// Mitsubishi GX Works2 project: LG Assembly 21-08-2019_F2   PLC: Q03UDV

PROGRAM MAIN
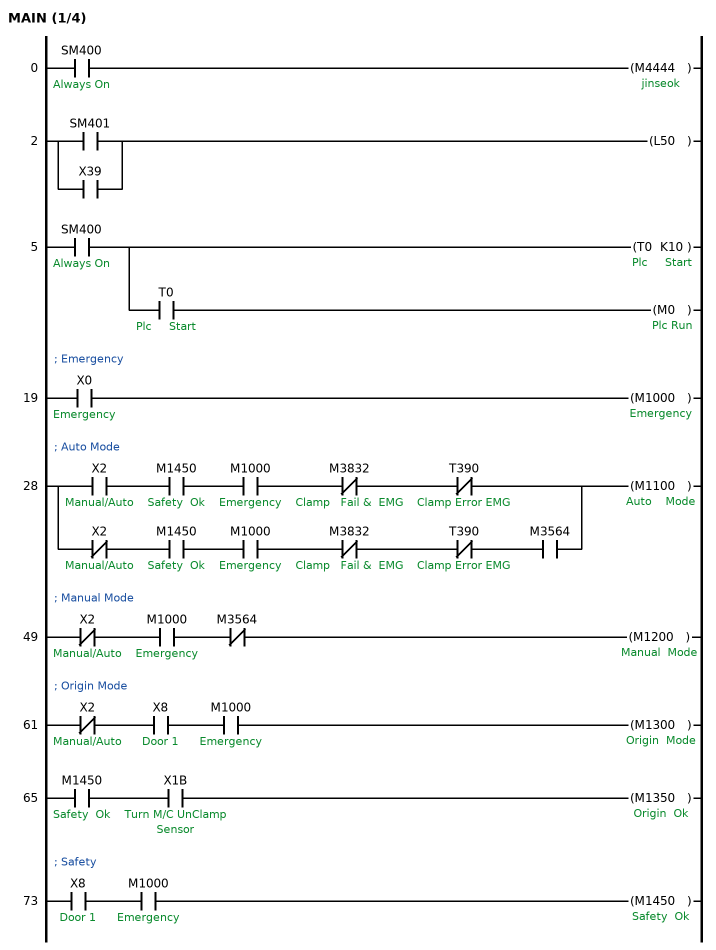
0     LD      SM400  ; Always On
      OUT     M4444  ; jinseok
2     LD      SM401
      OR      X39
      OUT     L50
5     LD      SM400  ; Always On
      OUT     T0 K10  ; Plc     Start
      AND     T0  ; Plc     Start
      OUT     M0  ; Plc Run
; Emergency
19    LD      X0  ; Emergency
      OUT     M1000  ; Emergency
; Auto Mode
28    LD      X2  ; Manual/Auto
      AND     M1450  ; Safety  Ok
      AND     M1000  ; Emergency
      ANI     M3832  ; Clamp   Fail &  EMG
      ANI     T390  ; Clamp Error EMG
      LDI     X2  ; Manual/Auto
      AND     M1450  ; Safety  Ok
      AND     M1000  ; Emergency
      ANI     M3832  ; Clamp   Fail &  EMG
      ANI     T390  ; Clamp Error EMG
      AND     M3564
      ORB
      OUT     M1100  ; Auto    Mode
; Manual Mode
49    LDI     X2  ; Manual/Auto
      AND     M1000  ; Emergency
      ANI     M3564
      OUT     M1200  ; Manual  Mode
; Origin Mode
61    LDI     X2  ; Manual/Auto
      AND     X8  ; Door 1
      AND     M1000  ; Emergency
      OUT     M1300  ; Origin  Mode
65    LD      M1450  ; Safety  Ok
      AND     X1B  ; Turn M/C UnClamp Sensor
      OUT     M1350  ; Origin  Ok
; Safety
73    LD      X8  ; Door 1
      AND     M1000  ; Emergency
      OUT     M1450  ; Safety  Ok
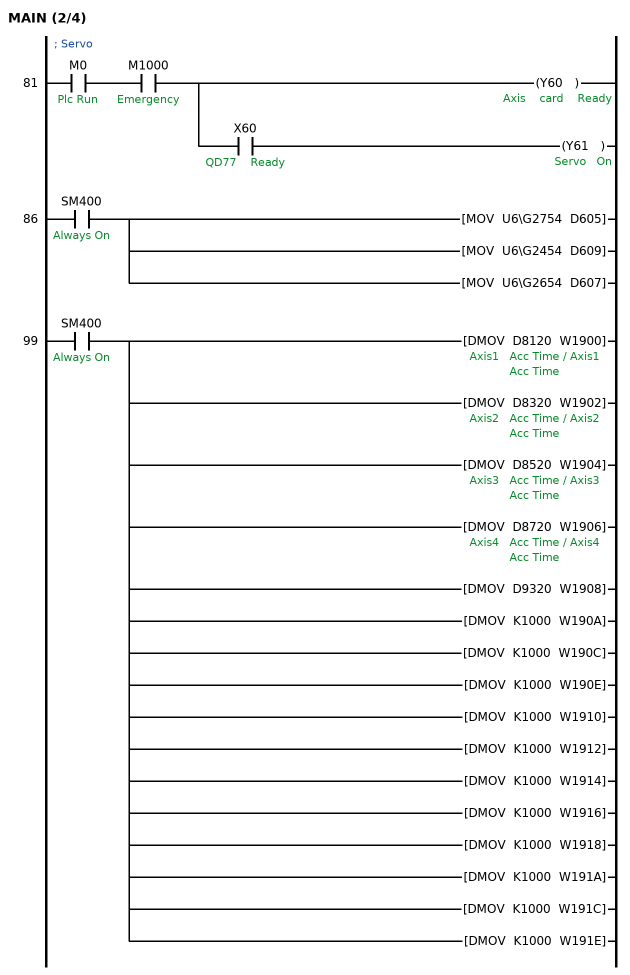
; Servo
81    LD      M0  ; Plc Run
      AND     M1000  ; Emergency
      OUT     Y60  ; Axis    card    Ready
      AND     X60  ; QD77    Ready
      OUT     Y61  ; Servo   On
86    LD      SM400  ; Always On
      MOV     U6\G2754 D605
      MOV     U6\G2454 D609
      MOV     U6\G2654 D607
99    LD      SM400  ; Always On
      DMOV    D8120 W1900  ; Axis1   Acc Time / Axis1   Acc Time
      DMOV    D8320 W1902  ; Axis2   Acc Time / Axis2   Acc Time
      DMOV    D8520 W1904  ; Axis3   Acc Time / Axis3   Acc Time
      DMOV    D8720 W1906  ; Axis4   Acc Time / Axis4   Acc Time
      DMOV    D9320 W1908
      DMOV    K1000 W190A
      DMOV    K1000 W190C
      DMOV    K1000 W190E
      DMOV    K1000 W1910
      DMOV    K1000 W1912
      DMOV    K1000 W1914
      DMOV    K1000 W1916
      DMOV    K1000 W1918
      DMOV    K1000 W191A
      DMOV    K1000 W191C
      DMOV    K1000 W191E
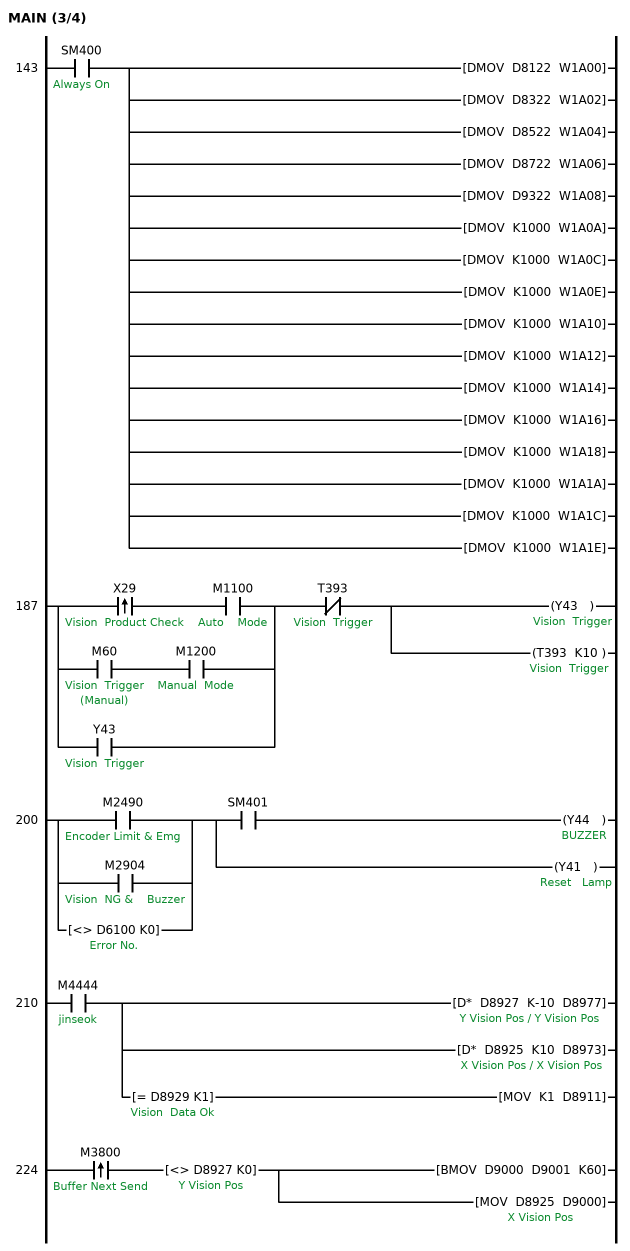
143   LD      SM400  ; Always On
      DMOV    D8122 W1A00
      DMOV    D8322 W1A02
      DMOV    D8522 W1A04
      DMOV    D8722 W1A06
      DMOV    D9322 W1A08
      DMOV    K1000 W1A0A
      DMOV    K1000 W1A0C
      DMOV    K1000 W1A0E
      DMOV    K1000 W1A10
      DMOV    K1000 W1A12
      DMOV    K1000 W1A14
      DMOV    K1000 W1A16
      DMOV    K1000 W1A18
      DMOV    K1000 W1A1A
      DMOV    K1000 W1A1C
      DMOV    K1000 W1A1E
187   LDP     X29  ; Vision  Product Check
      AND     M1100  ; Auto    Mode
      LD      M60  ; Vision  Trigger (Manual)
      AND     M1200  ; Manual  Mode
      ORB
      OR      Y43  ; Vision  Trigger
      ANI     T393  ; Vision  Trigger
      OUT     Y43  ; Vision  Trigger
      OUT     T393 K10  ; Vision  Trigger
200   LD      M2490  ; Encoder Limit & Emg
      OR      M2904  ; Vision  NG &    Buzzer
      OR<>    D6100 K0  ; Error No.
      MPS
      AND     SM401
      OUT     Y44  ; BUZZER
      MPP
      OUT     Y41  ; Reset   Lamp
210   LD      M4444  ; jinseok
      D*      D8927 K-10 D8977  ; Y Vision Pos / Y Vision Pos
      D*      D8925 K10 D8973  ; X Vision Pos / X Vision Pos
      AND=    D8929 K1  ; Vision  Data Ok
      MOV     K1 D8911
224   LDP     M3800  ; Buffer Next Send
      AND<>   D8927 K0  ; Y Vision Pos
      BMOV    D9000 D9001 K60
      MOV     D8925 D9000
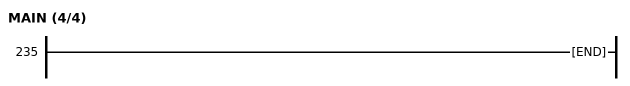
235   END
END_PROGRAM

PROGRAM ALARM
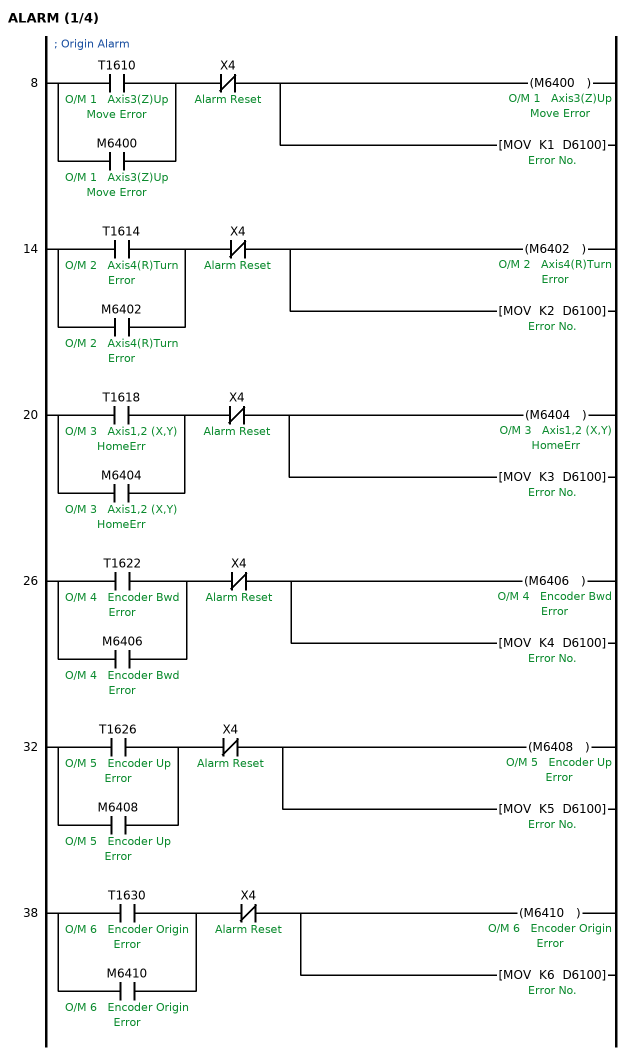
; Origin Alarm
8     LD      T1610  ; O/M 1   Axis3(Z)Up Move Error
      OR      M6400  ; O/M 1   Axis3(Z)Up Move Error
      ANI     X4  ; Alarm Reset
      OUT     M6400  ; O/M 1   Axis3(Z)Up Move Error
      MOV     K1 D6100  ; Error No.
14    LD      T1614  ; O/M 2   Axis4(R)Turn    Error
      OR      M6402  ; O/M 2   Axis4(R)Turn    Error
      ANI     X4  ; Alarm Reset
      OUT     M6402  ; O/M 2   Axis4(R)Turn    Error
      MOV     K2 D6100
20    LD      T1618  ; O/M 3   Axis1,2 (X,Y)   HomeErr
      OR      M6404  ; O/M 3   Axis1,2 (X,Y)   HomeErr
      ANI     X4  ; Alarm Reset
      OUT     M6404  ; O/M 3   Axis1,2 (X,Y)   HomeErr
      MOV     K3 D6100
26    LD      T1622  ; O/M 4   Encoder Bwd     Error
      OR      M6406  ; O/M 4   Encoder Bwd     Error
      ANI     X4  ; Alarm Reset
      OUT     M6406  ; O/M 4   Encoder Bwd     Error
      MOV     K4 D6100
32    LD      T1626  ; O/M 5   Encoder Up      Error
      OR      M6408  ; O/M 5   Encoder Up      Error
      ANI     X4  ; Alarm Reset
      OUT     M6408  ; O/M 5   Encoder Up      Error
      MOV     K5 D6100
38    LD      T1630  ; O/M 6   Encoder Origin  Error
      OR      M6410  ; O/M 6   Encoder Origin  Error
      ANI     X4  ; Alarm Reset
      OUT     M6410  ; O/M 6   Encoder Origin  Error
      MOV     K6 D6100
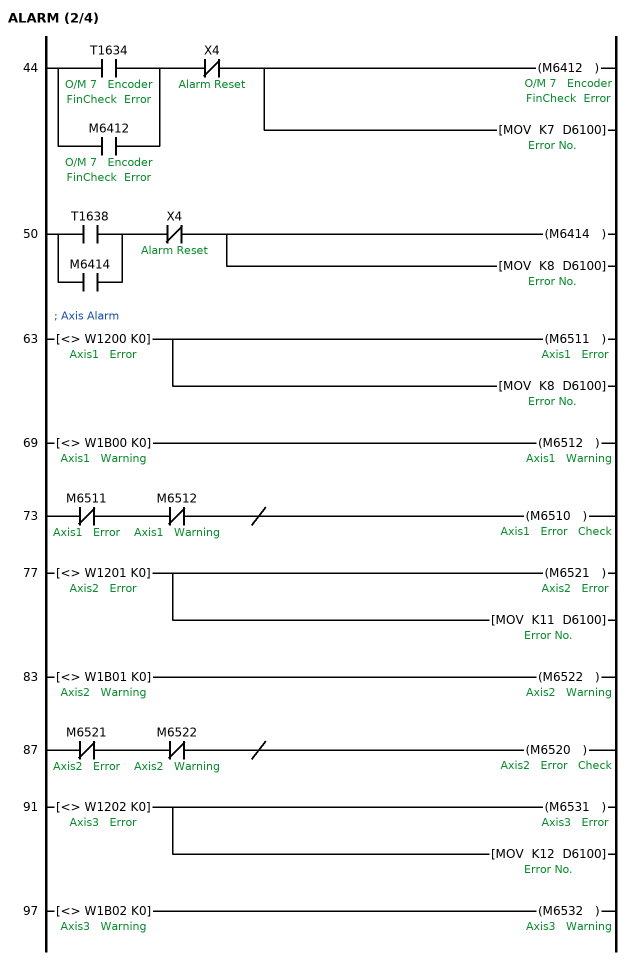
44    LD      T1634  ; O/M 7   Encoder FinCheck  Error
      OR      M6412  ; O/M 7   Encoder FinCheck  Error
      ANI     X4  ; Alarm Reset
      OUT     M6412  ; O/M 7   Encoder FinCheck  Error
      MOV     K7 D6100
50    LD      T1638
      OR      M6414
      ANI     X4  ; Alarm Reset
      OUT     M6414
      MOV     K8 D6100
; Axis Alarm
63    LD<>    W1200 K0  ; Axis1   Error
      OUT     M6511  ; Axis1   Error
      MOV     K8 D6100
69    LD<>    W1B00 K0  ; Axis1   Warning
      OUT     M6512  ; Axis1   Warning
73    LDI     M6511  ; Axis1   Error
      ANI     M6512  ; Axis1   Warning
      INV
      OUT     M6510  ; Axis1   Error   Check
77    LD<>    W1201 K0  ; Axis2   Error
      OUT     M6521  ; Axis2   Error
      MOV     K11 D6100
83    LD<>    W1B01 K0  ; Axis2   Warning
      OUT     M6522  ; Axis2   Warning
87    LDI     M6521  ; Axis2   Error
      ANI     M6522  ; Axis2   Warning
      INV
      OUT     M6520  ; Axis2   Error   Check
91    LD<>    W1202 K0  ; Axis3   Error
      OUT     M6531  ; Axis3   Error
      MOV     K12 D6100
97    LD<>    W1B02 K0  ; Axis3   Warning
      OUT     M6532  ; Axis3   Warning
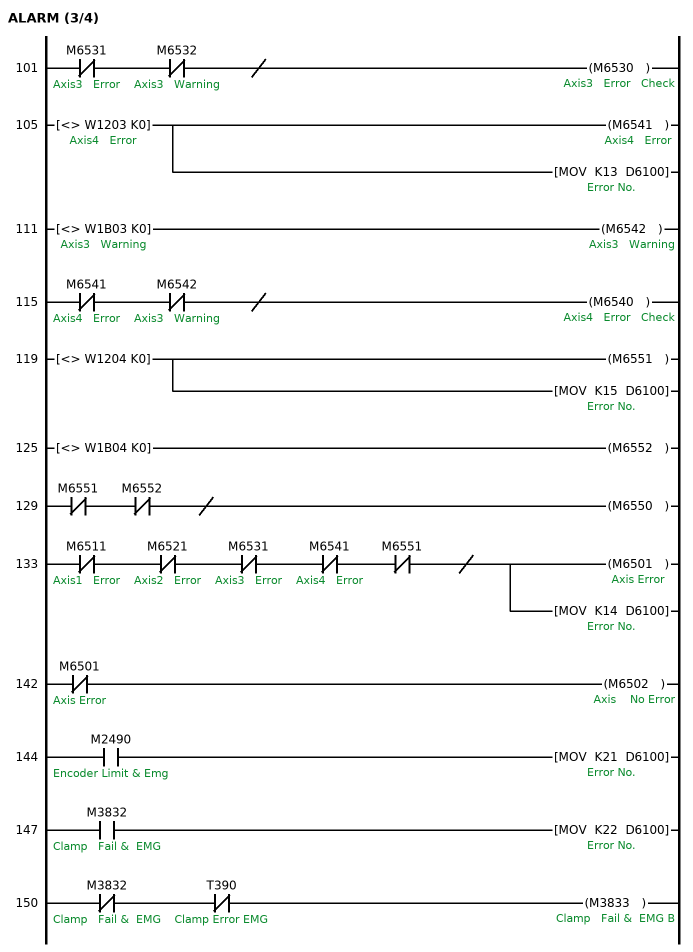
101   LDI     M6531  ; Axis3   Error
      ANI     M6532  ; Axis3   Warning
      INV
      OUT     M6530  ; Axis3   Error   Check
105   LD<>    W1203 K0  ; Axis4   Error
      OUT     M6541  ; Axis4   Error
      MOV     K13 D6100
111   LD<>    W1B03 K0  ; Axis3   Warning
      OUT     M6542  ; Axis3   Warning
115   LDI     M6541  ; Axis4   Error
      ANI     M6542  ; Axis3   Warning
      INV
      OUT     M6540  ; Axis4   Error   Check
119   LD<>    W1204 K0
      OUT     M6551
      MOV     K15 D6100
125   LD<>    W1B04 K0
      OUT     M6552
129   LDI     M6551
      ANI     M6552
      INV
      OUT     M6550
133   LDI     M6511  ; Axis1   Error
      ANI     M6521  ; Axis2   Error
      ANI     M6531  ; Axis3   Error
      ANI     M6541  ; Axis4   Error
      ANI     M6551
      INV
      OUT     M6501  ; Axis Error
      MOV     K14 D6100
142   LDI     M6501  ; Axis Error
      OUT     M6502  ; Axis    No Error
144   LD      M2490  ; Encoder Limit & Emg
      MOV     K21 D6100
147   LD      M3832  ; Clamp   Fail &  EMG
      MOV     K22 D6100
150   LDI     M3832  ; Clamp   Fail &  EMG
      ANI     T390  ; Clamp Error EMG
      OUT     M3833  ; Clamp   Fail &  EMG B
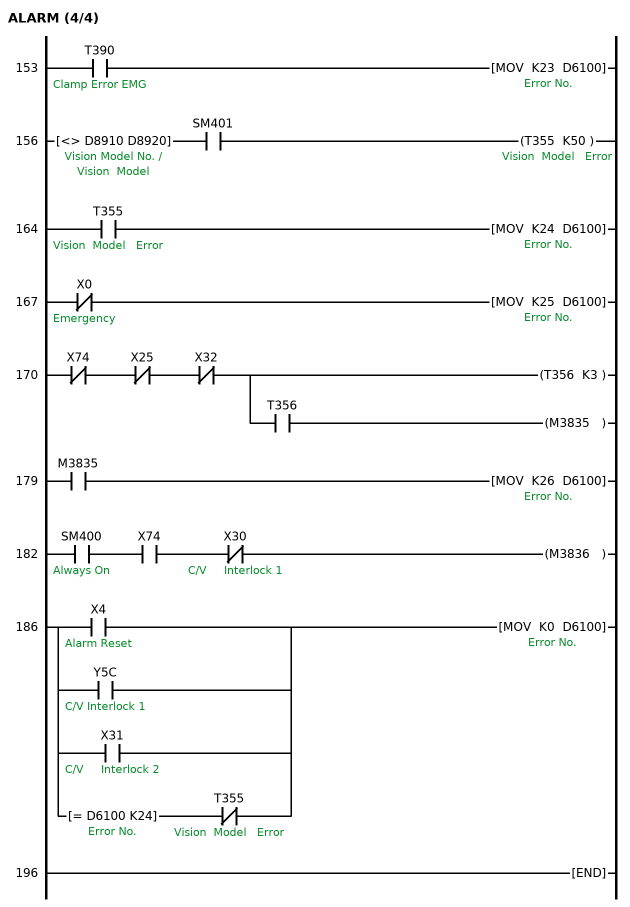
153   LD      T390  ; Clamp Error EMG
      MOV     K23 D6100
156   LD<>    D8910 D8920  ; Vision Model No. / Vision  Model
      AND     SM401
      OUT     T355 K50  ; Vision  Model   Error
164   LD      T355  ; Vision  Model   Error
      MOV     K24 D6100
167   LDI     X0  ; Emergency
      MOV     K25 D6100
170   LDI     X74
      ANI     X25
      ANI     X32
      OUT     T356 K3
      AND     T356
      OUT     M3835
179   LD      M3835
      MOV     K26 D6100
182   LD      SM400  ; Always On
      AND     X74
      ANI     X30  ; C/V     Interlock 1
      OUT     M3836
186   LD      X4  ; Alarm Reset
      OR      Y5C  ; C/V Interlock 1
      OR      X31  ; C/V     Interlock 2
      LD=     D6100 K24  ; Error No.
      ANI     T355  ; Vision  Model   Error
      ORB
      MOV     K0 D6100
196   END
END_PROGRAM

PROGRAM AUTO
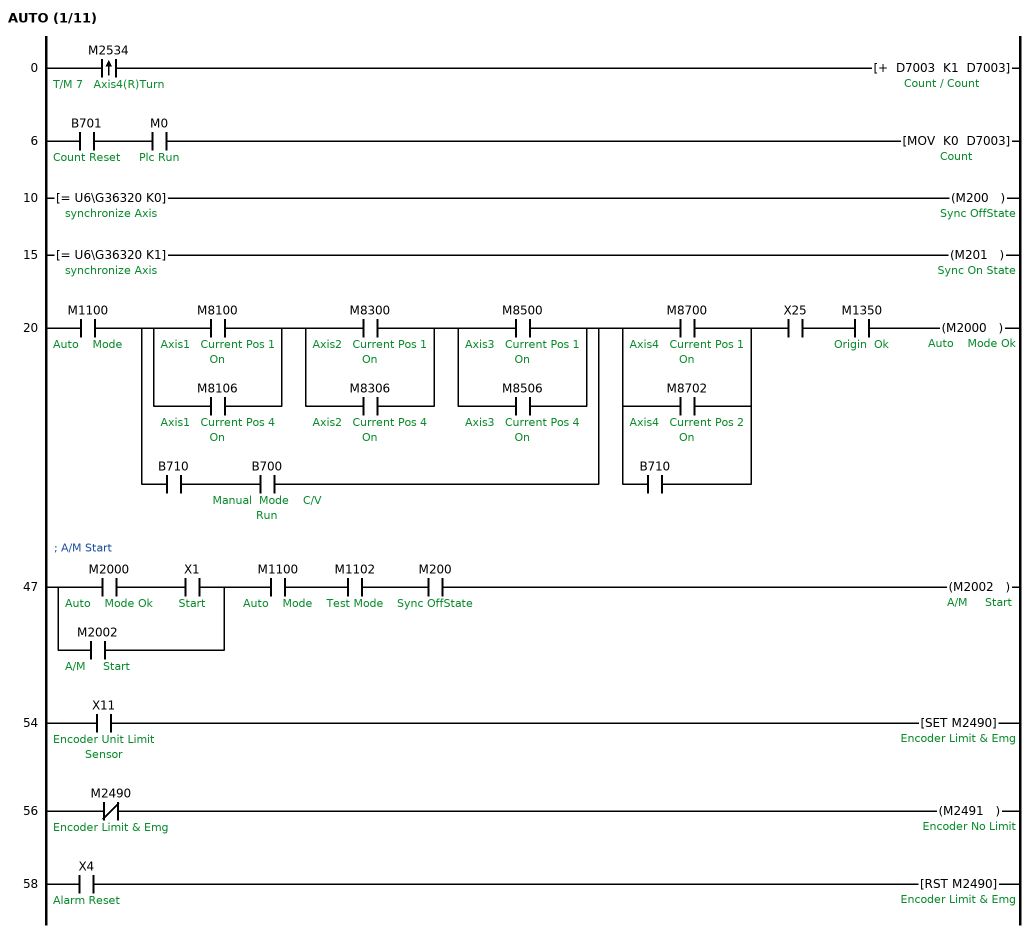
0     LDP     M2534  ; T/M 7   Axis4(R)Turn
      +       D7003 K1 D7003  ; Count
6     LD      B701  ; Count Reset
      AND     M0  ; Plc Run
      MOV     K0 D7003
10    LD=     U6\G36320 K0  ; synchronize Axis
      OUT     M200  ; Sync OffState
15    LD=     U6\G36320 K1  ; synchronize Axis
      OUT     M201  ; Sync On State
20    LD      M1100  ; Auto    Mode
      LD      M8100  ; Axis1   Current Pos 1 On
      OR      M8106  ; Axis1   Current Pos 4 On
      LD      M8300  ; Axis2   Current Pos 1 On
      OR      M8306  ; Axis2   Current Pos 4 On
      ANB
      LD      M8500  ; Axis3   Current Pos 1 On
      OR      M8506  ; Axis3   Current Pos 4 On
      ANB
      LD      B710
      AND     B700  ; Manual  Mode    C/V Run
      ORB
      ANB
      LD      M8700  ; Axis4   Current Pos 1 On
      OR      M8702  ; Axis4   Current Pos 2 On
      OR      B710
      ANB
      AND     X25
      AND     M1350  ; Origin  Ok
      OUT     M2000  ; Auto    Mode Ok
; A/M Start
47    LD      M2000  ; Auto    Mode Ok
      AND     X1  ; Start
      OR      M2002  ; A/M     Start
      AND     M1100  ; Auto    Mode
      AND     M1102  ; Test Mode
      AND     M200  ; Sync OffState
      OUT     M2002  ; A/M     Start
54    LD      X11  ; Encoder Unit Limit Sensor
      SET     M2490  ; Encoder Limit & Emg
56    LDI     M2490  ; Encoder Limit & Emg
      OUT     M2491  ; Encoder No Limit
58    LD      X4  ; Alarm Reset
      RST     M2490  ; Encoder Limit & Emg
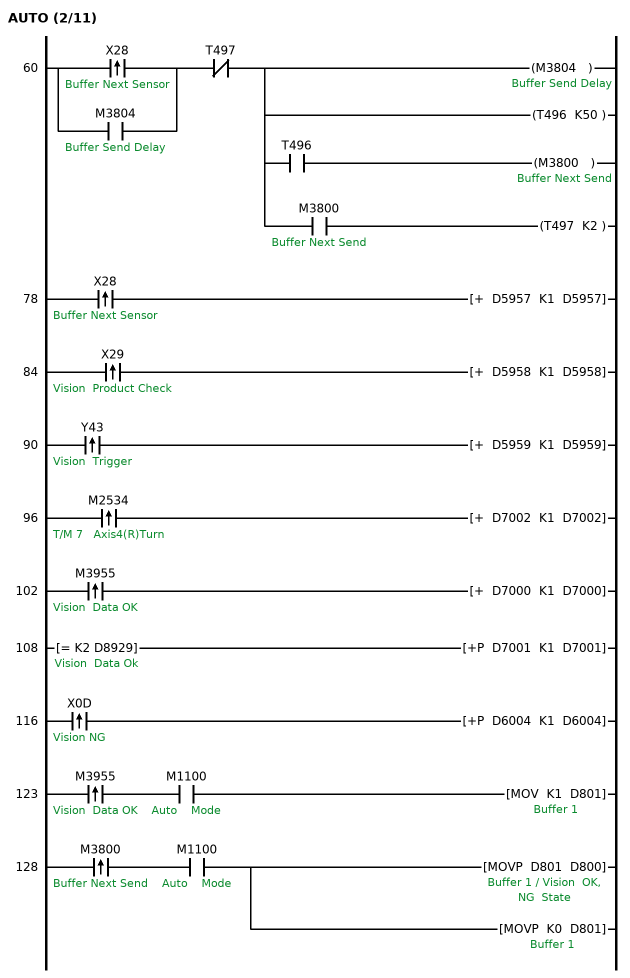
60    LDP     X28  ; Buffer Next Sensor
      OR      M3804  ; Buffer Send Delay
      ANI     T497
      OUT     M3804  ; Buffer Send Delay
      OUT     T496 K50
      MPS
      AND     T496
      OUT     M3800  ; Buffer Next Send
      MPP
      AND     M3800  ; Buffer Next Send
      OUT     T497 K2
78    LDP     X28  ; Buffer Next Sensor
      +       D5957 K1 D5957
84    LDP     X29  ; Vision  Product Check
      +       D5958 K1 D5958
90    LDP     Y43  ; Vision  Trigger
      +       D5959 K1 D5959
96    LDP     M2534  ; T/M 7   Axis4(R)Turn
      +       D7002 K1 D7002
102   LDP     M3955  ; Vision  Data OK
      +       D7000 K1 D7000
108   LD=     K2 D8929  ; Vision  Data Ok
      +P      D7001 K1 D7001
116   LDP     X0D  ; Vision NG
      +P      D6004 K1 D6004
123   LDP     M3955  ; Vision  Data OK
      AND     M1100  ; Auto    Mode
      MOV     K1 D801  ; Buffer 1
128   LDP     M3800  ; Buffer Next Send
      AND     M1100  ; Auto    Mode
      MOVP    D801 D800  ; Vision  OK, NG  State
      MOVP    K0 D801
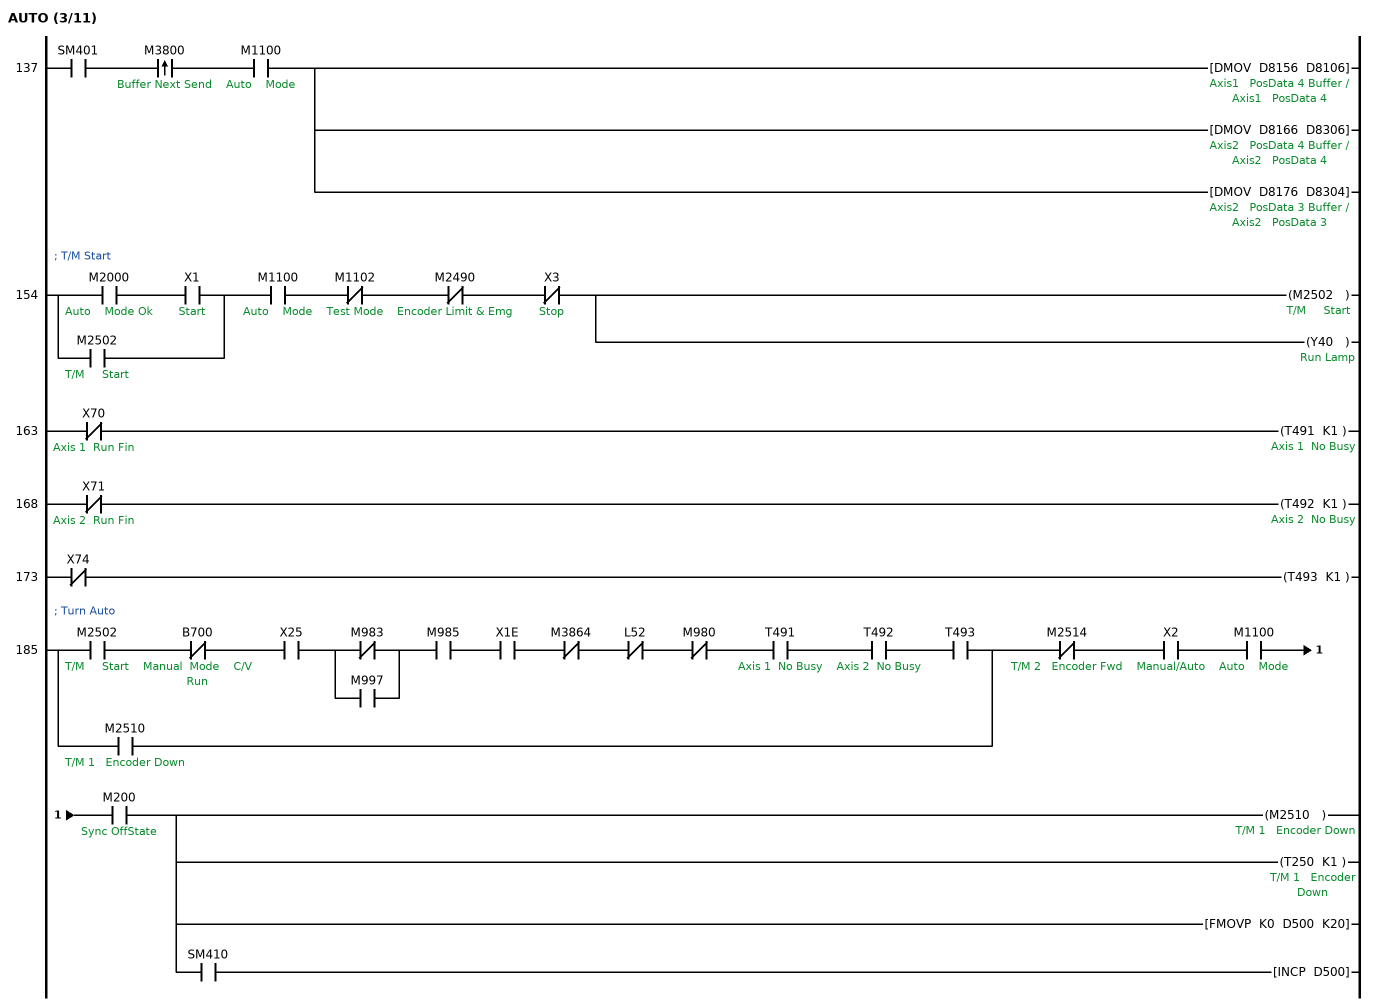
137   LD      SM401
      ANDP    M3800  ; Buffer Next Send
      AND     M1100  ; Auto    Mode
      DMOV    D8156 D8106  ; Axis1   PosData 4 Buffer / Axis1   PosData 4
      DMOV    D8166 D8306  ; Axis2   PosData 4 Buffer / Axis2   PosData 4
      DMOV    D8176 D8304  ; Axis2   PosData 3 Buffer / Axis2   PosData 3
; T/M Start
154   LD      M2000  ; Auto    Mode Ok
      AND     X1  ; Start
      OR      M2502  ; T/M     Start
      AND     M1100  ; Auto    Mode
      ANI     M1102  ; Test Mode
      ANI     M2490  ; Encoder Limit & Emg
      ANI     X3  ; Stop
      OUT     M2502  ; T/M     Start
      OUT     Y40  ; Run Lamp
163   LDI     X70  ; Axis 1  Run Fin
      OUT     T491 K1  ; Axis 1  No Busy
168   LDI     X71  ; Axis 2  Run Fin
      OUT     T492 K1  ; Axis 2  No Busy
173   LDI     X74
      OUT     T493 K1
; Turn Auto
185   LD      M2502  ; T/M     Start
      ANI     B700  ; Manual  Mode    C/V Run
      AND     X25
      LDI     M983
      OR      M997
      ANB
      AND     M985
      AND     X1E
      ANI     M3864
      ANI     L52
      ANI     M980
      AND     T491  ; Axis 1  No Busy
      AND     T492  ; Axis 2  No Busy
      AND     T493
      OR      M2510  ; T/M 1   Encoder Down
      ANI     M2514  ; T/M 2   Encoder Fwd
      AND     X2  ; Manual/Auto
      AND     M1100  ; Auto    Mode
      AND     M200  ; Sync OffState
      OUT     M2510  ; T/M 1   Encoder Down
      OUT     T250 K1  ; T/M 1   Encoder Down
      FMOVP   K0 D500 K20
      AND     SM410
      INCP    D500
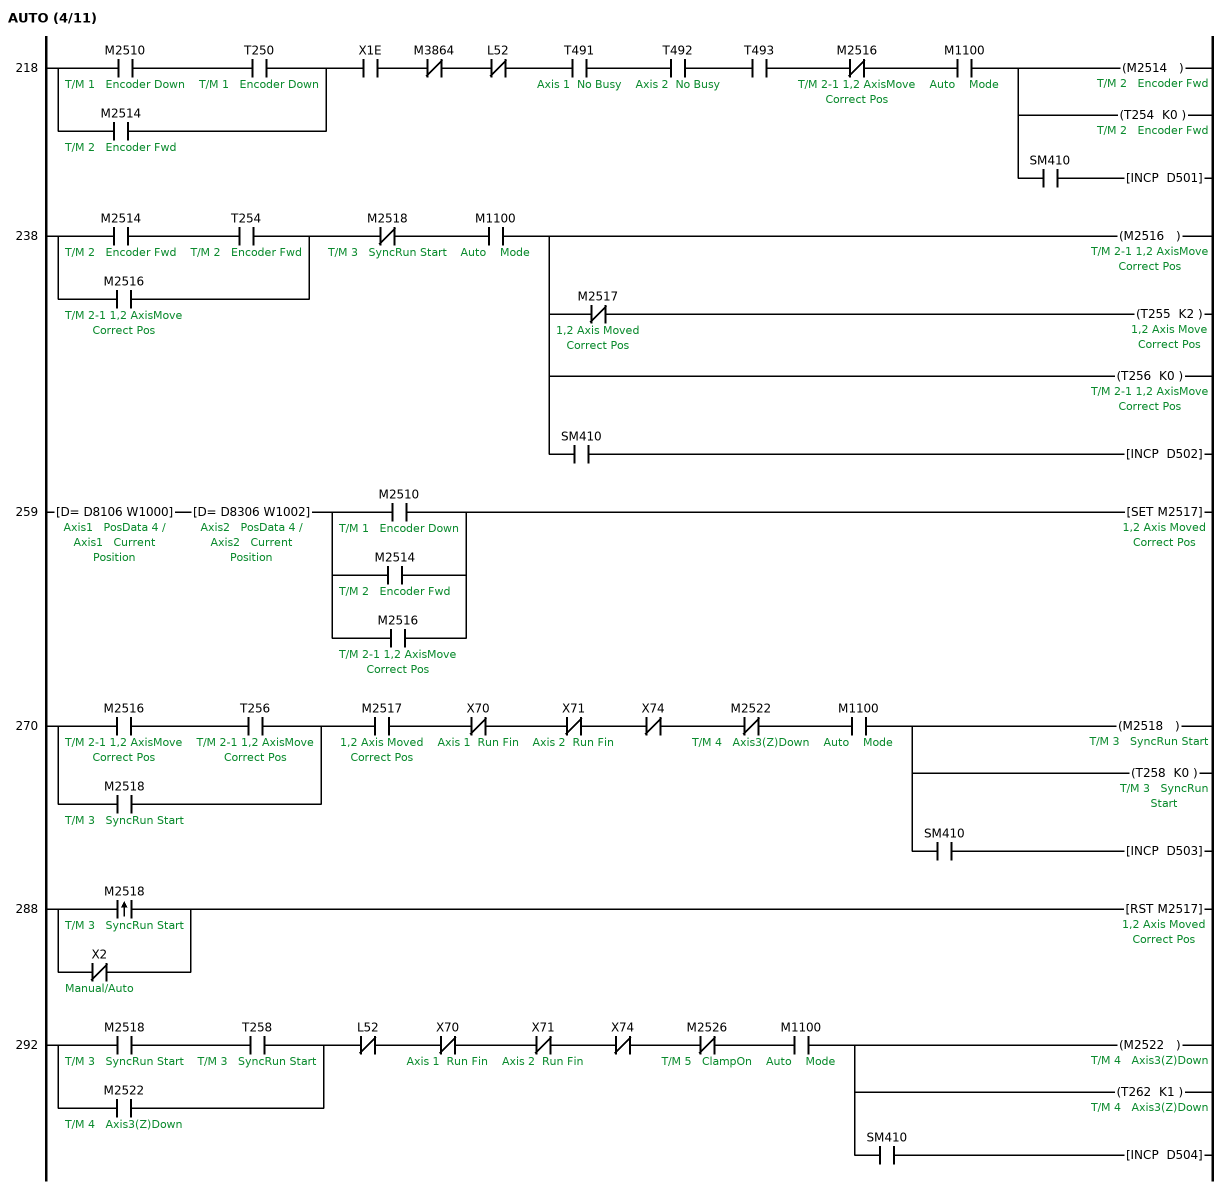
218   LD      M2510  ; T/M 1   Encoder Down
      AND     T250  ; T/M 1   Encoder Down
      OR      M2514  ; T/M 2   Encoder Fwd
      AND     X1E
      ANI     M3864
      ANI     L52
      AND     T491  ; Axis 1  No Busy
      AND     T492  ; Axis 2  No Busy
      AND     T493
      ANI     M2516  ; T/M 2-1 1,2 AxisMove Correct Pos
      AND     M1100  ; Auto    Mode
      OUT     M2514  ; T/M 2   Encoder Fwd
      OUT     T254 K0  ; T/M 2   Encoder Fwd
      AND     SM410
      INCP    D501
238   LD      M2514  ; T/M 2   Encoder Fwd
      AND     T254  ; T/M 2   Encoder Fwd
      OR      M2516  ; T/M 2-1 1,2 AxisMove Correct Pos
      ANI     M2518  ; T/M 3   SyncRun Start
      AND     M1100  ; Auto    Mode
      OUT     M2516  ; T/M 2-1 1,2 AxisMove Correct Pos
      MPS
      ANI     M2517  ; 1,2 Axis Moved Correct Pos
      OUT     T255 K2  ; 1,2 Axis Move Correct Pos
      MPP
      OUT     T256 K0  ; T/M 2-1 1,2 AxisMove Correct Pos
      AND     SM410
      INCP    D502
259   LDD=    D8106 W1000  ; Axis1   PosData 4 / Axis1   Current Position
      ANDD=   D8306 W1002  ; Axis2   PosData 4 / Axis2   Current Position
      LD      M2510  ; T/M 1   Encoder Down
      OR      M2514  ; T/M 2   Encoder Fwd
      OR      M2516  ; T/M 2-1 1,2 AxisMove Correct Pos
      ANB
      SET     M2517  ; 1,2 Axis Moved Correct Pos
270   LD      M2516  ; T/M 2-1 1,2 AxisMove Correct Pos
      AND     T256  ; T/M 2-1 1,2 AxisMove Correct Pos
      OR      M2518  ; T/M 3   SyncRun Start
      AND     M2517  ; 1,2 Axis Moved Correct Pos
      ANI     X70  ; Axis 1  Run Fin
      ANI     X71  ; Axis 2  Run Fin
      ANI     X74
      ANI     M2522  ; T/M 4   Axis3(Z)Down
      AND     M1100  ; Auto    Mode
      OUT     M2518  ; T/M 3   SyncRun Start
      OUT     T258 K0  ; T/M 3   SyncRun Start
      AND     SM410
      INCP    D503
288   LDP     M2518  ; T/M 3   SyncRun Start
      ORI     X2  ; Manual/Auto
      RST     M2517  ; 1,2 Axis Moved Correct Pos
292   LD      M2518  ; T/M 3   SyncRun Start
      AND     T258  ; T/M 3   SyncRun Start
      OR      M2522  ; T/M 4   Axis3(Z)Down
      ANI     L52
      ANI     X70  ; Axis 1  Run Fin
      ANI     X71  ; Axis 2  Run Fin
      ANI     X74
      ANI     M2526  ; T/M 5   ClampOn
      AND     M1100  ; Auto    Mode
      OUT     M2522  ; T/M 4   Axis3(Z)Down
      OUT     T262 K1  ; T/M 4   Axis3(Z)Down
      AND     SM410
      INCP    D504
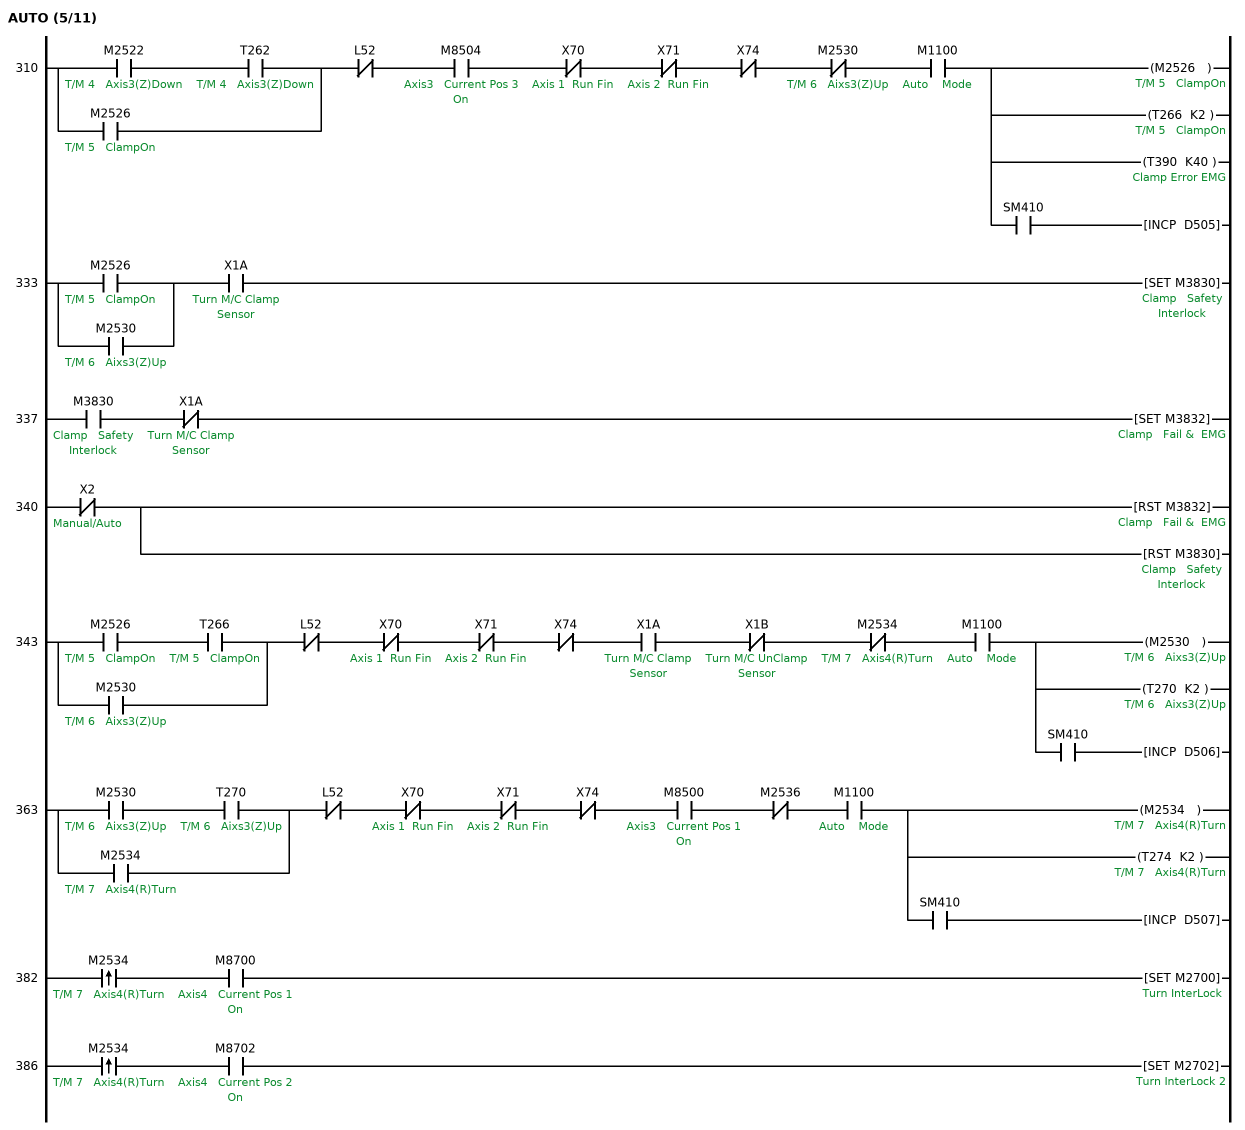
310   LD      M2522  ; T/M 4   Axis3(Z)Down
      AND     T262  ; T/M 4   Axis3(Z)Down
      OR      M2526  ; T/M 5   ClampOn
      ANI     L52
      AND     M8504  ; Axis3   Current Pos 3 On
      ANI     X70  ; Axis 1  Run Fin
      ANI     X71  ; Axis 2  Run Fin
      ANI     X74
      ANI     M2530  ; T/M 6   Aixs3(Z)Up
      AND     M1100  ; Auto    Mode
      OUT     M2526  ; T/M 5   ClampOn
      OUT     T266 K2  ; T/M 5   ClampOn
      OUT     T390 K40  ; Clamp Error EMG
      AND     SM410
      INCP    D505
333   LD      M2526  ; T/M 5   ClampOn
      OR      M2530  ; T/M 6   Aixs3(Z)Up
      AND     X1A  ; Turn M/C Clamp Sensor
      SET     M3830  ; Clamp   Safety  Interlock
337   LD      M3830  ; Clamp   Safety  Interlock
      ANI     X1A  ; Turn M/C Clamp Sensor
      SET     M3832  ; Clamp   Fail &  EMG
340   LDI     X2  ; Manual/Auto
      RST     M3832  ; Clamp   Fail &  EMG
      RST     M3830  ; Clamp   Safety  Interlock
343   LD      M2526  ; T/M 5   ClampOn
      AND     T266  ; T/M 5   ClampOn
      OR      M2530  ; T/M 6   Aixs3(Z)Up
      ANI     L52
      ANI     X70  ; Axis 1  Run Fin
      ANI     X71  ; Axis 2  Run Fin
      ANI     X74
      AND     X1A  ; Turn M/C Clamp Sensor
      ANI     X1B  ; Turn M/C UnClamp Sensor
      ANI     M2534  ; T/M 7   Axis4(R)Turn
      AND     M1100  ; Auto    Mode
      OUT     M2530  ; T/M 6   Aixs3(Z)Up
      OUT     T270 K2  ; T/M 6   Aixs3(Z)Up
      AND     SM410
      INCP    D506
363   LD      M2530  ; T/M 6   Aixs3(Z)Up
      AND     T270  ; T/M 6   Aixs3(Z)Up
      OR      M2534  ; T/M 7   Axis4(R)Turn
      ANI     L52
      ANI     X70  ; Axis 1  Run Fin
      ANI     X71  ; Axis 2  Run Fin
      ANI     X74
      AND     M8500  ; Axis3   Current Pos 1 On
      ANI     M2536
      AND     M1100  ; Auto    Mode
      OUT     M2534  ; T/M 7   Axis4(R)Turn
      OUT     T274 K2  ; T/M 7   Axis4(R)Turn
      AND     SM410
      INCP    D507
382   LDP     M2534  ; T/M 7   Axis4(R)Turn
      AND     M8700  ; Axis4   Current Pos 1 On
      SET     M2700  ; Turn InterLock
386   LDP     M2534  ; T/M 7   Axis4(R)Turn
      AND     M8702  ; Axis4   Current Pos 2 On
      SET     M2702  ; Turn InterLock 2
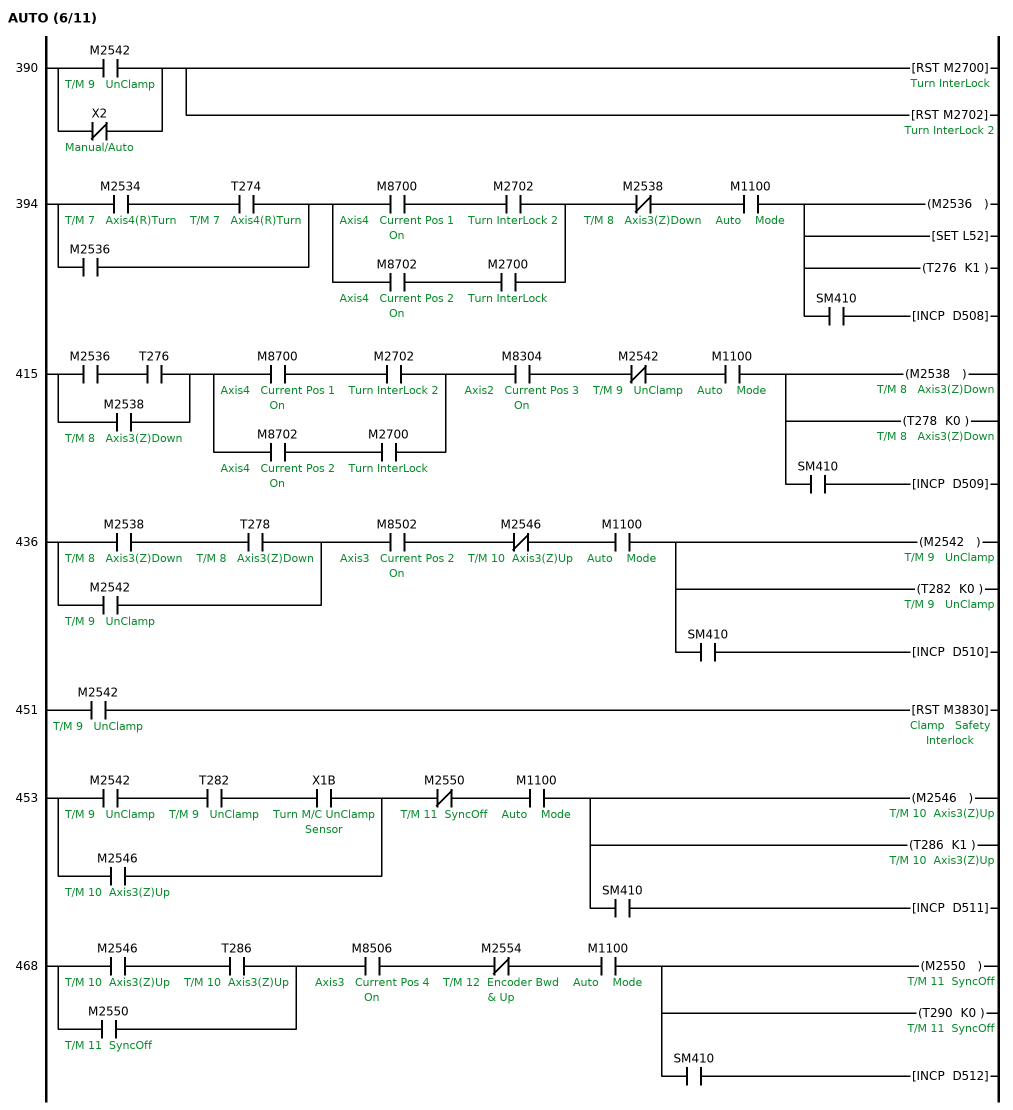
390   LD      M2542  ; T/M 9   UnClamp
      ORI     X2  ; Manual/Auto
      RST     M2700  ; Turn InterLock
      RST     M2702  ; Turn InterLock 2
394   LD      M2534  ; T/M 7   Axis4(R)Turn
      AND     T274  ; T/M 7   Axis4(R)Turn
      OR      M2536
      LD      M8700  ; Axis4   Current Pos 1 On
      AND     M2702  ; Turn InterLock 2
      LD      M8702  ; Axis4   Current Pos 2 On
      AND     M2700  ; Turn InterLock
      ORB
      ANB
      ANI     M2538  ; T/M 8   Axis3(Z)Down
      AND     M1100  ; Auto    Mode
      OUT     M2536
      SET     L52
      OUT     T276 K1
      AND     SM410
      INCP    D508
415   LD      M2536
      AND     T276
      OR      M2538  ; T/M 8   Axis3(Z)Down
      LD      M8700  ; Axis4   Current Pos 1 On
      AND     M2702  ; Turn InterLock 2
      LD      M8702  ; Axis4   Current Pos 2 On
      AND     M2700  ; Turn InterLock
      ORB
      ANB
      AND     M8304  ; Axis2   Current Pos 3 On
      ANI     M2542  ; T/M 9   UnClamp
      AND     M1100  ; Auto    Mode
      OUT     M2538  ; T/M 8   Axis3(Z)Down
      OUT     T278 K0  ; T/M 8   Axis3(Z)Down
      AND     SM410
      INCP    D509
436   LD      M2538  ; T/M 8   Axis3(Z)Down
      AND     T278  ; T/M 8   Axis3(Z)Down
      OR      M2542  ; T/M 9   UnClamp
      AND     M8502  ; Axis3   Current Pos 2 On
      ANI     M2546  ; T/M 10  Axis3(Z)Up
      AND     M1100  ; Auto    Mode
      OUT     M2542  ; T/M 9   UnClamp
      OUT     T282 K0  ; T/M 9   UnClamp
      AND     SM410
      INCP    D510
451   LD      M2542  ; T/M 9   UnClamp
      RST     M3830  ; Clamp   Safety  Interlock
453   LD      M2542  ; T/M 9   UnClamp
      AND     T282  ; T/M 9   UnClamp
      AND     X1B  ; Turn M/C UnClamp Sensor
      OR      M2546  ; T/M 10  Axis3(Z)Up
      ANI     M2550  ; T/M 11  SyncOff
      AND     M1100  ; Auto    Mode
      OUT     M2546  ; T/M 10  Axis3(Z)Up
      OUT     T286 K1  ; T/M 10  Axis3(Z)Up
      AND     SM410
      INCP    D511
468   LD      M2546  ; T/M 10  Axis3(Z)Up
      AND     T286  ; T/M 10  Axis3(Z)Up
      OR      M2550  ; T/M 11  SyncOff
      AND     M8506  ; Axis3   Current Pos 4 On
      ANI     M2554  ; T/M 12  Encoder Bwd & Up
      AND     M1100  ; Auto    Mode
      OUT     M2550  ; T/M 11  SyncOff
      OUT     T290 K0  ; T/M 11  SyncOff
      AND     SM410
      INCP    D512
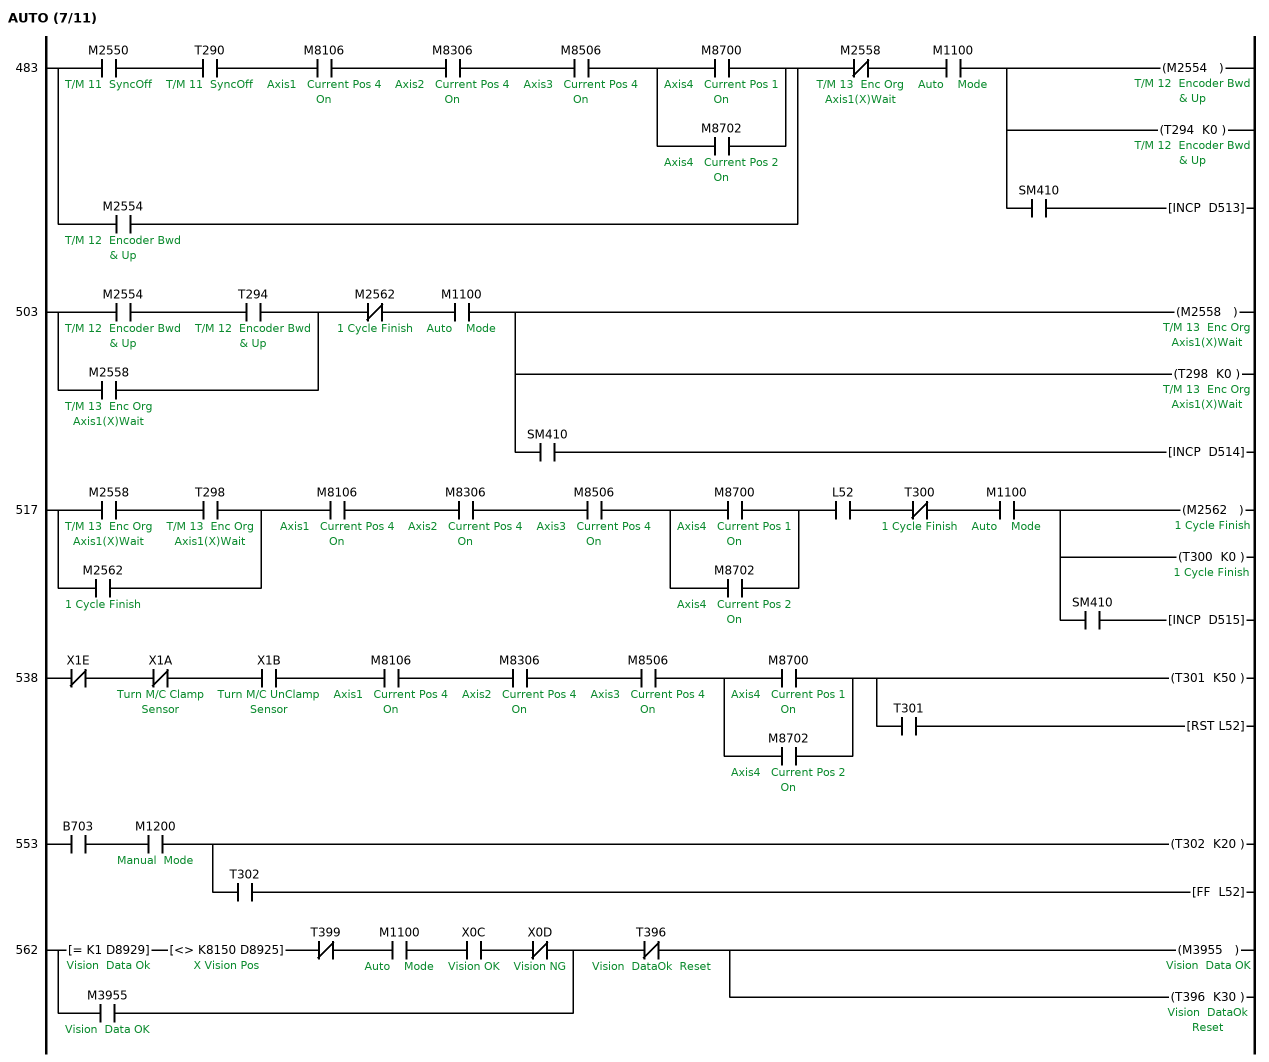
483   LD      M2550  ; T/M 11  SyncOff
      AND     T290  ; T/M 11  SyncOff
      AND     M8106  ; Axis1   Current Pos 4 On
      AND     M8306  ; Axis2   Current Pos 4 On
      AND     M8506  ; Axis3   Current Pos 4 On
      LD      M8700  ; Axis4   Current Pos 1 On
      OR      M8702  ; Axis4   Current Pos 2 On
      ANB
      OR      M2554  ; T/M 12  Encoder Bwd & Up
      ANI     M2558  ; T/M 13  Enc Org Axis1(X)Wait
      AND     M1100  ; Auto    Mode
      OUT     M2554  ; T/M 12  Encoder Bwd & Up
      OUT     T294 K0  ; T/M 12  Encoder Bwd & Up
      AND     SM410
      INCP    D513
503   LD      M2554  ; T/M 12  Encoder Bwd & Up
      AND     T294  ; T/M 12  Encoder Bwd & Up
      OR      M2558  ; T/M 13  Enc Org Axis1(X)Wait
      ANI     M2562  ; 1 Cycle Finish
      AND     M1100  ; Auto    Mode
      OUT     M2558  ; T/M 13  Enc Org Axis1(X)Wait
      OUT     T298 K0  ; T/M 13  Enc Org Axis1(X)Wait
      AND     SM410
      INCP    D514
517   LD      M2558  ; T/M 13  Enc Org Axis1(X)Wait
      AND     T298  ; T/M 13  Enc Org Axis1(X)Wait
      OR      M2562  ; 1 Cycle Finish
      AND     M8106  ; Axis1   Current Pos 4 On
      AND     M8306  ; Axis2   Current Pos 4 On
      AND     M8506  ; Axis3   Current Pos 4 On
      LD      M8700  ; Axis4   Current Pos 1 On
      OR      M8702  ; Axis4   Current Pos 2 On
      ANB
      AND     L52
      ANI     T300  ; 1 Cycle Finish
      AND     M1100  ; Auto    Mode
      OUT     M2562  ; 1 Cycle Finish
      OUT     T300 K0  ; 1 Cycle Finish
      AND     SM410
      INCP    D515
538   LDI     X1E
      ANI     X1A  ; Turn M/C Clamp Sensor
      AND     X1B  ; Turn M/C UnClamp Sensor
      AND     M8106  ; Axis1   Current Pos 4 On
      AND     M8306  ; Axis2   Current Pos 4 On
      AND     M8506  ; Axis3   Current Pos 4 On
      LD      M8700  ; Axis4   Current Pos 1 On
      OR      M8702  ; Axis4   Current Pos 2 On
      ANB
      OUT     T301 K50
      AND     T301
      RST     L52
553   LD      B703
      AND     M1200  ; Manual  Mode
      OUT     T302 K20
      AND     T302
      FF      L52
562   LD=     K1 D8929  ; Vision  Data Ok
      AND<>   K8150 D8925  ; X Vision Pos
      ANI     T399
      AND     M1100  ; Auto    Mode
      AND     X0C  ; Vision OK
      ANI     X0D  ; Vision NG
      OR      M3955  ; Vision  Data OK
      ANI     T396  ; Vision  DataOk  Reset
      OUT     M3955  ; Vision  Data OK
      OUT     T396 K30  ; Vision  DataOk  Reset
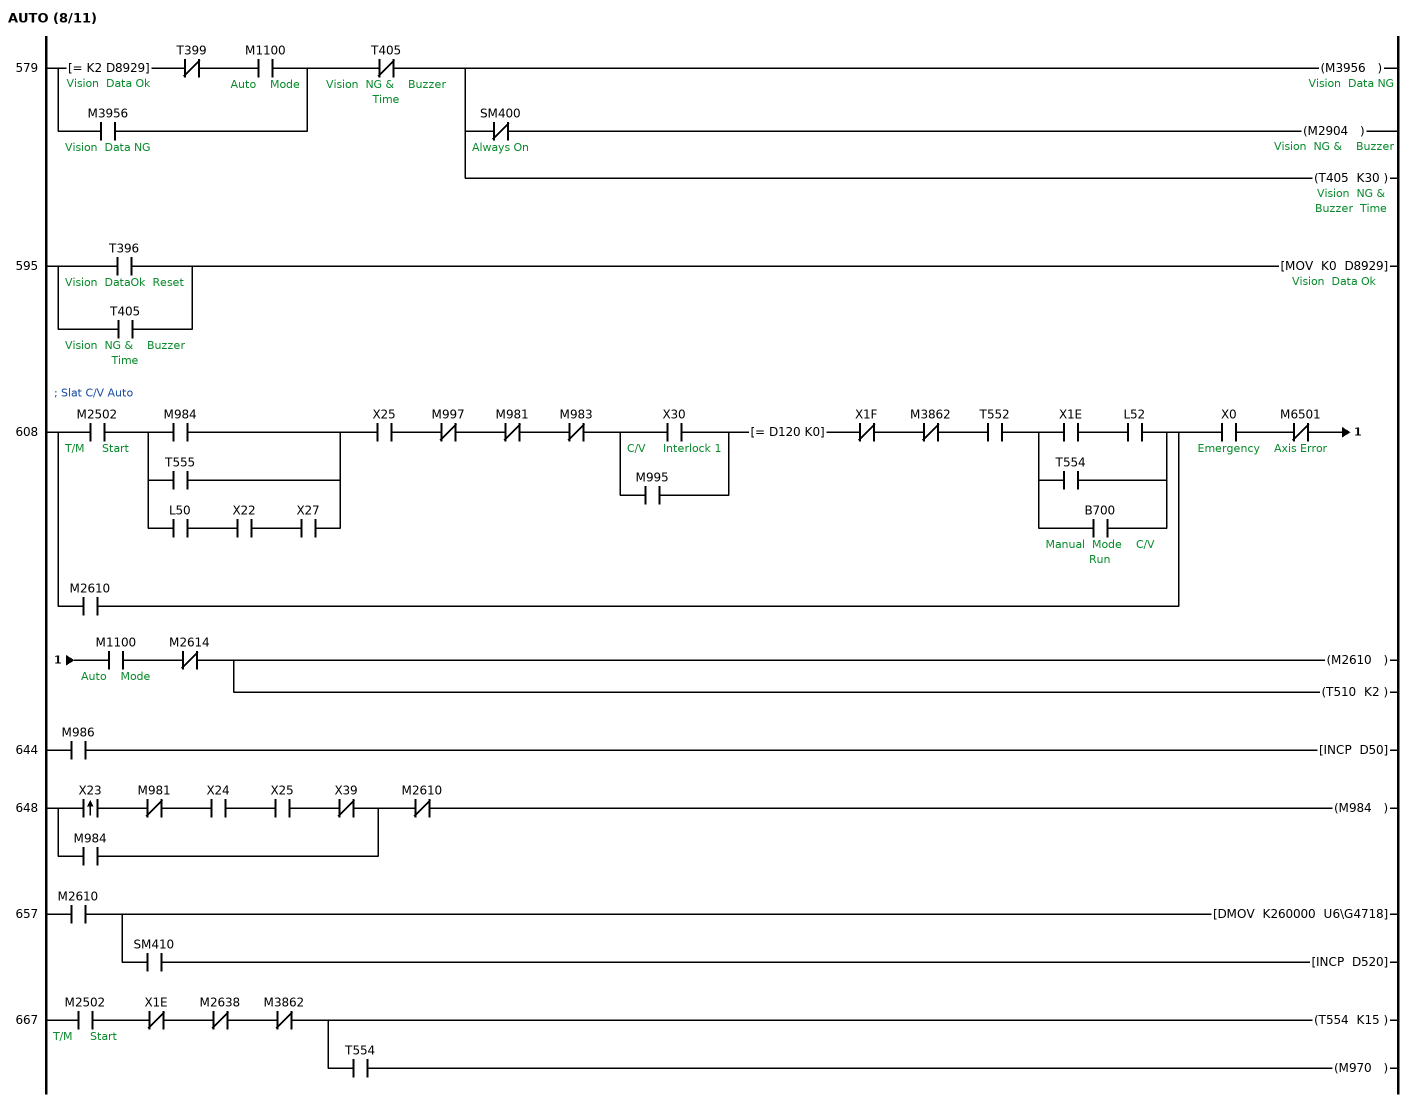
579   LD=     K2 D8929  ; Vision  Data Ok
      ANI     T399
      AND     M1100  ; Auto    Mode
      OR      M3956  ; Vision  Data NG
      ANI     T405  ; Vision  NG &    Buzzer  Time
      OUT     M3956  ; Vision  Data NG
      MPS
      ANI     SM400  ; Always On
      OUT     M2904  ; Vision  NG &    Buzzer
      MPP
      OUT     T405 K30  ; Vision  NG &    Buzzer  Time
595   LD      T396  ; Vision  DataOk  Reset
      OR      T405  ; Vision  NG &    Buzzer  Time
      MOV     K0 D8929
; Slat C/V Auto
608   LD      M2502  ; T/M     Start
      LD      M984
      OR      T555
      LD      L50
      AND     X22
      AND     X27
      ORB
      ANB
      AND     X25
      ANI     M997
      ANI     M981
      ANI     M983
      LD      X30  ; C/V     Interlock 1
      OR      M995
      ANB
      AND=    D120 K0
      ANI     X1F
      ANI     M3862
      AND     T552
      LD      X1E
      AND     L52
      OR      T554
      OR      B700  ; Manual  Mode    C/V Run
      ANB
      OR      M2610
      AND     X0  ; Emergency
      ANI     M6501  ; Axis Error
      AND     M1100  ; Auto    Mode
      ANI     M2614
      OUT     M2610
      OUT     T510 K2
644   LD      M986
      INCP    D50
648   LDP     X23
      ANI     M981
      AND     X24
      AND     X25
      ANI     X39
      OR      M984
      ANI     M2610
      OUT     M984
657   LD      M2610
      DMOV    K260000 U6\G4718
      AND     SM410
      INCP    D520
667   LD      M2502  ; T/M     Start
      ANI     X1E
      ANI     M2638
      ANI     M3862
      OUT     T554 K15
      AND     T554
      OUT     M970
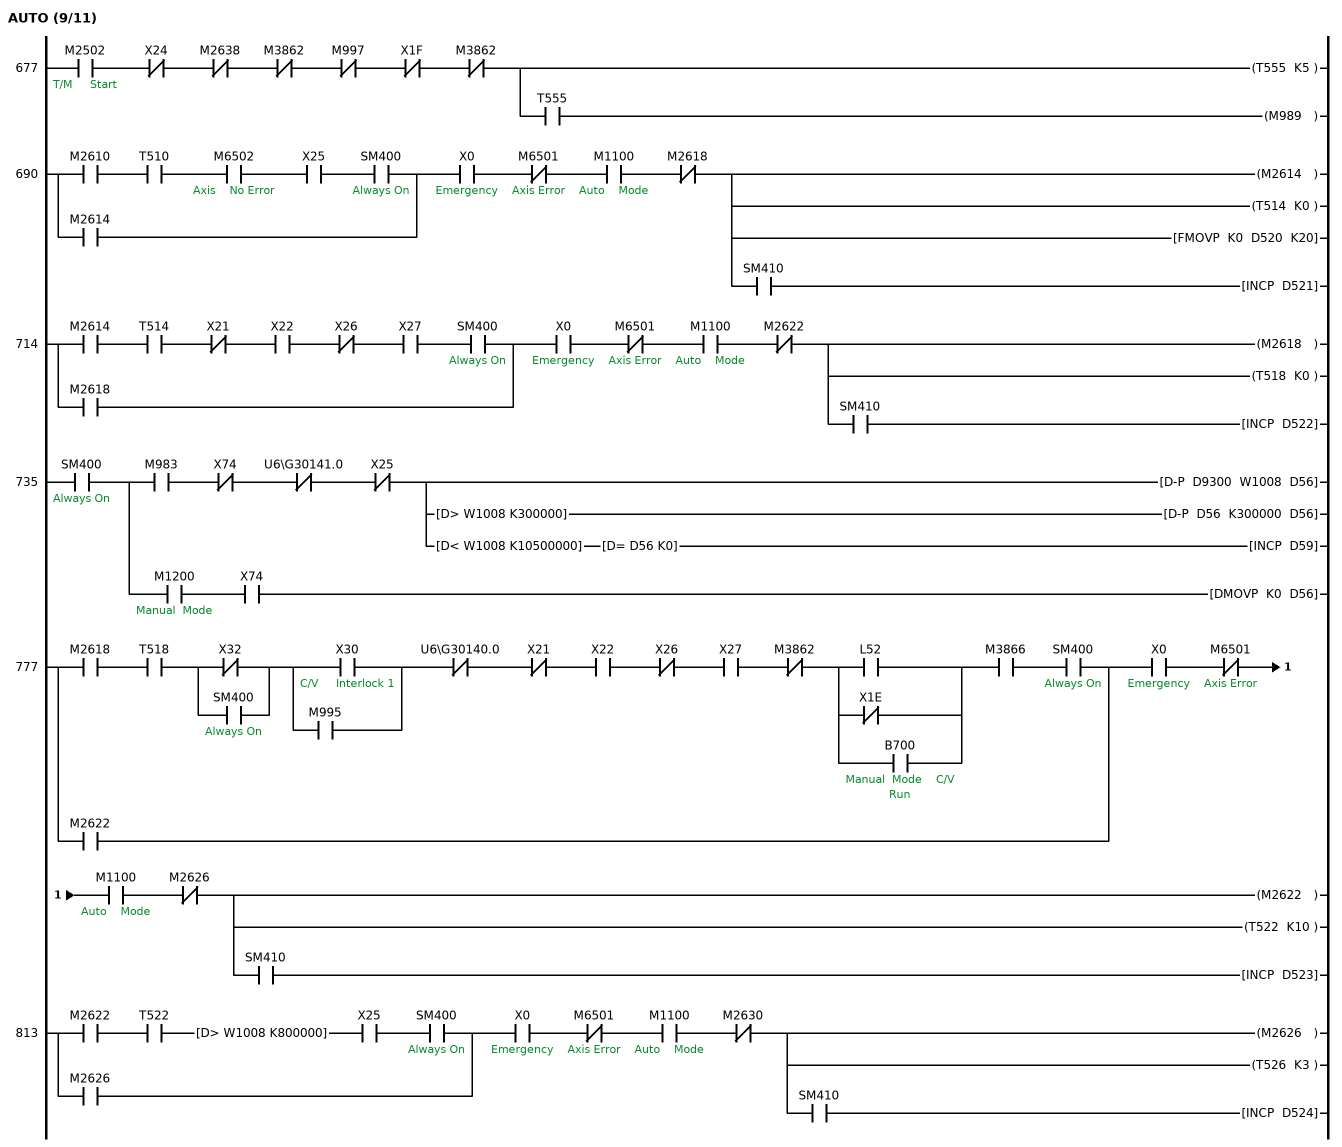
677   LD      M2502  ; T/M     Start
      ANI     X24
      ANI     M2638
      ANI     M3862
      ANI     M997
      ANI     X1F
      ANI     M3862
      OUT     T555 K5
      AND     T555
      OUT     M989
690   LD      M2610
      AND     T510
      AND     M6502  ; Axis    No Error
      AND     X25
      AND     SM400  ; Always On
      OR      M2614
      AND     X0  ; Emergency
      ANI     M6501  ; Axis Error
      AND     M1100  ; Auto    Mode
      ANI     M2618
      OUT     M2614
      OUT     T514 K0
      FMOVP   K0 D520 K20
      AND     SM410
      INCP    D521
714   LD      M2614
      AND     T514
      ANI     X21
      AND     X22
      ANI     X26
      AND     X27
      AND     SM400  ; Always On
      OR      M2618
      AND     X0  ; Emergency
      ANI     M6501  ; Axis Error
      AND     M1100  ; Auto    Mode
      ANI     M2622
      OUT     M2618
      OUT     T518 K0
      AND     SM410
      INCP    D522
735   LD      SM400  ; Always On
      MPS
      AND     M983
      ANI     X74
      ANI     U6\G30141.0
      ANI     X25
      D-P     D9300 W1008 D56
      MPS
      ANDD>   W1008 K300000
      D-P     D56 K300000 D56
      MPP
      ANDD<   W1008 K10500000
      ANDD=   D56 K0
      INCP    D59
      MPP
      AND     M1200  ; Manual  Mode
      AND     X74
      DMOVP   K0 D56
777   LD      M2618
      AND     T518
      LDI     X32
      OR      SM400  ; Always On
      ANB
      LD      X30  ; C/V     Interlock 1
      OR      M995
      ANB
      ANI     U6\G30140.0
      ANI     X21
      AND     X22
      ANI     X26
      AND     X27
      ANI     M3862
      LD      L52
      ORI     X1E
      OR      B700  ; Manual  Mode    C/V Run
      ANB
      AND     M3866
      AND     SM400  ; Always On
      OR      M2622
      AND     X0  ; Emergency
      ANI     M6501  ; Axis Error
      AND     M1100  ; Auto    Mode
      ANI     M2626
      OUT     M2622
      OUT     T522 K10
      AND     SM410
      INCP    D523
813   LD      M2622
      AND     T522
      ANDD>   W1008 K800000
      AND     X25
      AND     SM400  ; Always On
      OR      M2626
      AND     X0  ; Emergency
      ANI     M6501  ; Axis Error
      AND     M1100  ; Auto    Mode
      ANI     M2630
      OUT     M2626
      OUT     T526 K3
      AND     SM410
      INCP    D524
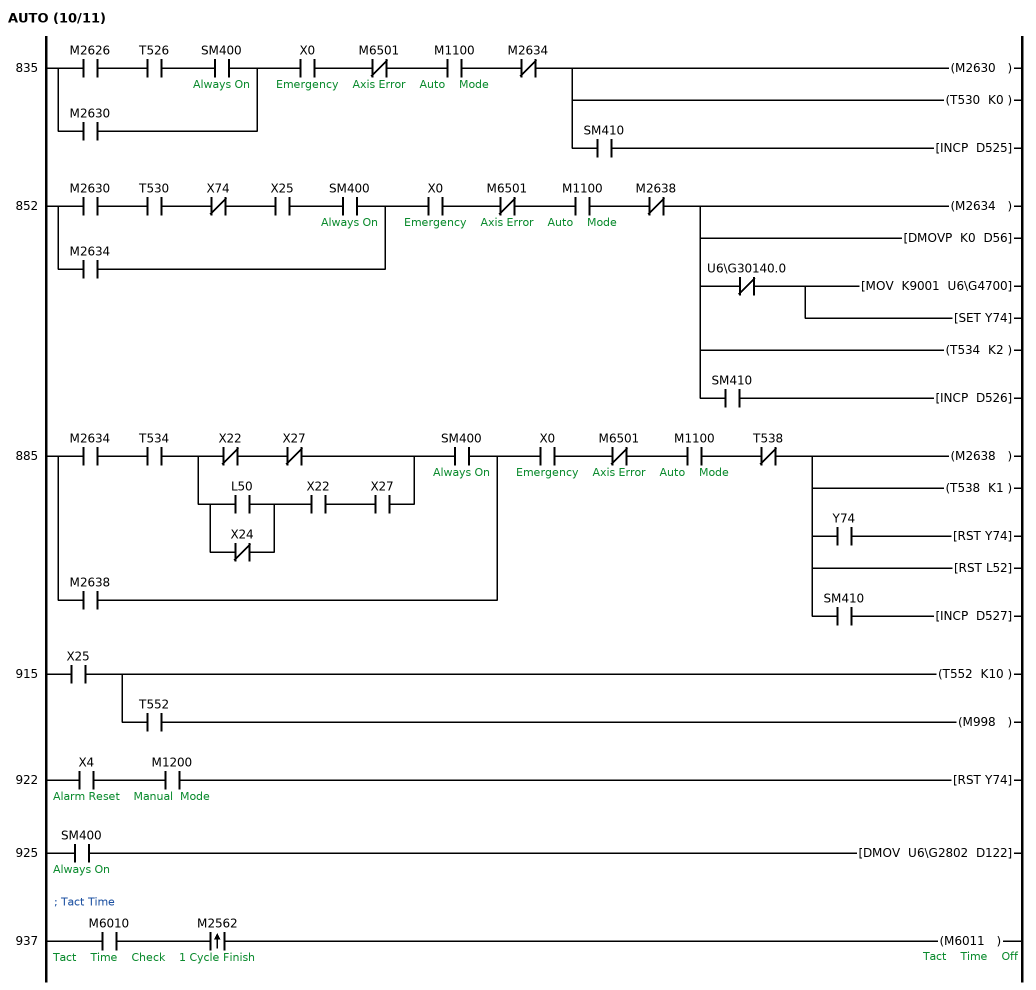
835   LD      M2626
      AND     T526
      AND     SM400  ; Always On
      OR      M2630
      AND     X0  ; Emergency
      ANI     M6501  ; Axis Error
      AND     M1100  ; Auto    Mode
      ANI     M2634
      OUT     M2630
      OUT     T530 K0
      AND     SM410
      INCP    D525
852   LD      M2630
      AND     T530
      ANI     X74
      AND     X25
      AND     SM400  ; Always On
      OR      M2634
      AND     X0  ; Emergency
      ANI     M6501  ; Axis Error
      AND     M1100  ; Auto    Mode
      ANI     M2638
      OUT     M2634
      DMOVP   K0 D56
      MPS
      ANI     U6\G30140.0
      MOV     K9001 U6\G4700
      SET     Y74
      MPP
      OUT     T534 K2
      AND     SM410
      INCP    D526
885   LD      M2634
      AND     T534
      LDI     X22
      ANI     X27
      LD      L50
      ORI     X24
      AND     X22
      AND     X27
      ORB
      ANB
      AND     SM400  ; Always On
      OR      M2638
      AND     X0  ; Emergency
      ANI     M6501  ; Axis Error
      AND     M1100  ; Auto    Mode
      ANI     T538
      OUT     M2638
      OUT     T538 K1
      MPS
      AND     Y74
      RST     Y74
      MPP
      RST     L52
      AND     SM410
      INCP    D527
915   LD      X25
      OUT     T552 K10
      AND     T552
      OUT     M998
922   LD      X4  ; Alarm Reset
      AND     M1200  ; Manual  Mode
      RST     Y74
925   LD      SM400  ; Always On
      DMOV    U6\G2802 D122
; Tact Time
937   LD      M6010  ; Tact    Time    Check
      ANDP    M2562  ; 1 Cycle Finish
      OUT     M6011  ; Tact    Time    Off
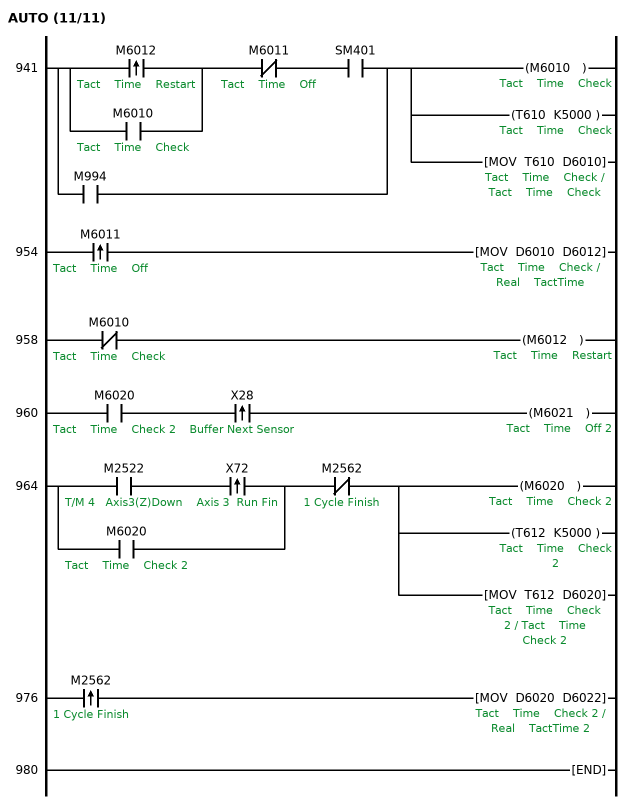
941   LDP     M6012  ; Tact    Time    Restart
      OR      M6010  ; Tact    Time    Check
      ANI     M6011  ; Tact    Time    Off
      AND     SM401
      OR      M994
      OUT     M6010  ; Tact    Time    Check
      OUT     T610 K5000  ; Tact    Time    Check
      MOV     T610 D6010  ; Tact    Time    Check
954   LDP     M6011  ; Tact    Time    Off
      MOV     D6010 D6012  ; Real    TactTime
958   LDI     M6010  ; Tact    Time    Check
      OUT     M6012  ; Tact    Time    Restart
960   LD      M6020  ; Tact    Time    Check 2
      ANDP    X28  ; Buffer Next Sensor
      OUT     M6021  ; Tact    Time    Off 2
964   LD      M2522  ; T/M 4   Axis3(Z)Down
      ANDP    X72  ; Axis 3  Run Fin
      OR      M6020  ; Tact    Time    Check 2
      ANI     M2562  ; 1 Cycle Finish
      OUT     M6020  ; Tact    Time    Check 2
      OUT     T612 K5000  ; Tact    Time    Check 2
      MOV     T612 D6020  ; Tact    Time    Check 2
976   LDP     M2562  ; 1 Cycle Finish
      MOV     D6020 D6022  ; Real    TactTime 2
980   END
END_PROGRAM

PROGRAM CONSTDAT
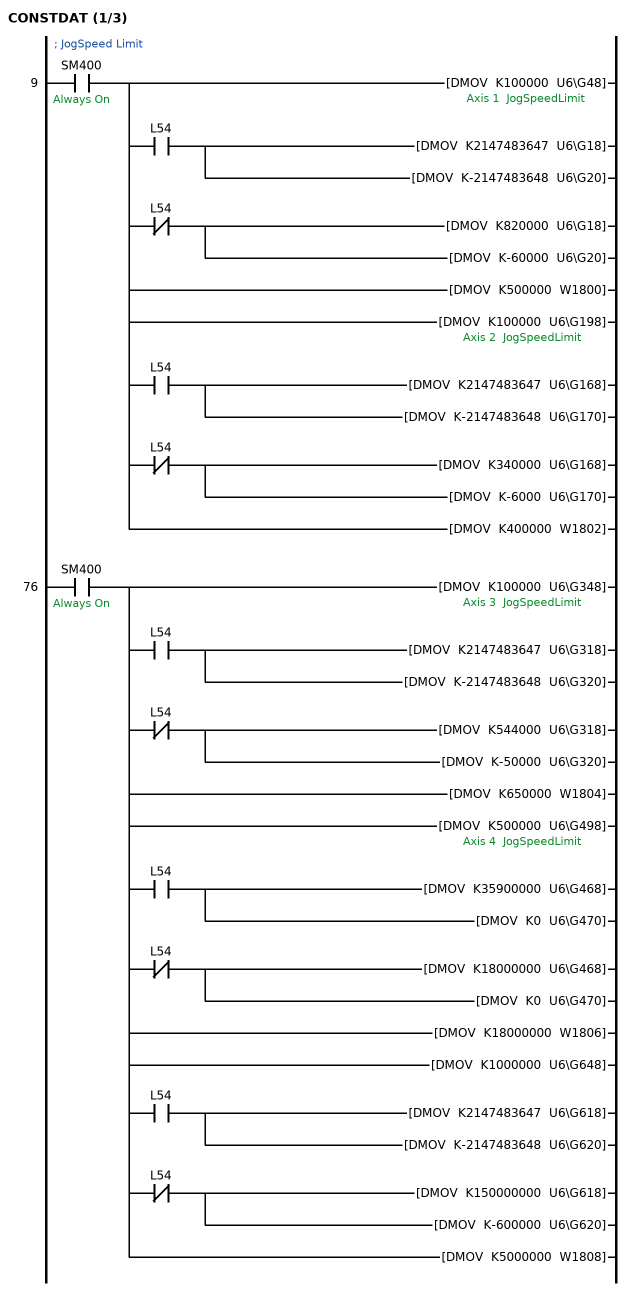
; JogSpeed Limit
9     LD      SM400  ; Always On
      DMOV    K100000 U6\G48  ; Axis 1  JogSpeedLimit
      MPS
      AND     L54
      DMOV    K2147483647 U6\G18
      DMOV    K-2147483648 U6\G20
      MRD
      ANI     L54
      DMOV    K820000 U6\G18
      DMOV    K-60000 U6\G20
      MPP
      DMOV    K500000 W1800
      DMOV    K100000 U6\G198  ; Axis 2  JogSpeedLimit
      MPS
      AND     L54
      DMOV    K2147483647 U6\G168
      DMOV    K-2147483648 U6\G170
      MRD
      ANI     L54
      DMOV    K340000 U6\G168
      DMOV    K-6000 U6\G170
      MPP
      DMOV    K400000 W1802
76    LD      SM400  ; Always On
      DMOV    K100000 U6\G348  ; Axis 3  JogSpeedLimit
      MPS
      AND     L54
      DMOV    K2147483647 U6\G318
      DMOV    K-2147483648 U6\G320
      MRD
      ANI     L54
      DMOV    K544000 U6\G318
      DMOV    K-50000 U6\G320
      MPP
      DMOV    K650000 W1804
      DMOV    K500000 U6\G498  ; Axis 4  JogSpeedLimit
      MPS
      AND     L54
      DMOV    K35900000 U6\G468
      DMOV    K0 U6\G470
      MRD
      ANI     L54
      DMOV    K18000000 U6\G468
      DMOV    K0 U6\G470
      MPP
      DMOV    K18000000 W1806
      DMOV    K1000000 U6\G648
      MPS
      AND     L54
      DMOV    K2147483647 U6\G618
      DMOV    K-2147483648 U6\G620
      MRD
      ANI     L54
      DMOV    K150000000 U6\G618
      DMOV    K-600000 U6\G620
      MPP
      DMOV    K5000000 W1808
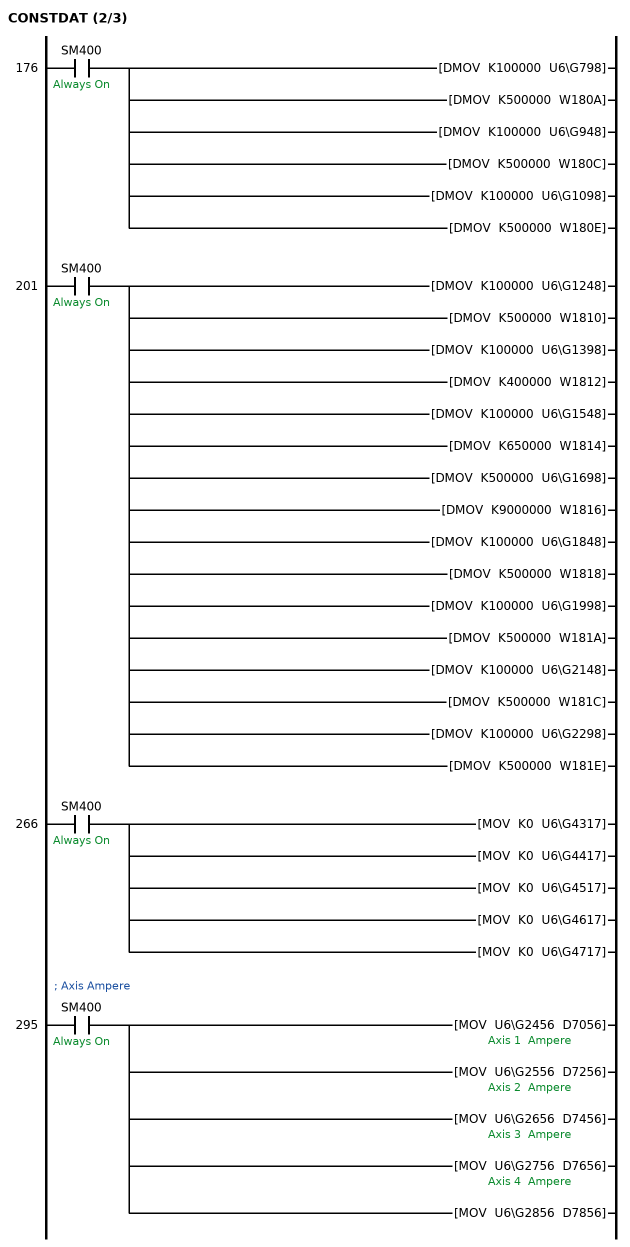
176   LD      SM400  ; Always On
      DMOV    K100000 U6\G798
      DMOV    K500000 W180A
      DMOV    K100000 U6\G948
      DMOV    K500000 W180C
      DMOV    K100000 U6\G1098
      DMOV    K500000 W180E
201   LD      SM400  ; Always On
      DMOV    K100000 U6\G1248
      DMOV    K500000 W1810
      DMOV    K100000 U6\G1398
      DMOV    K400000 W1812
      DMOV    K100000 U6\G1548
      DMOV    K650000 W1814
      DMOV    K500000 U6\G1698
      DMOV    K9000000 W1816
      DMOV    K100000 U6\G1848
      DMOV    K500000 W1818
      DMOV    K100000 U6\G1998
      DMOV    K500000 W181A
      DMOV    K100000 U6\G2148
      DMOV    K500000 W181C
      DMOV    K100000 U6\G2298
      DMOV    K500000 W181E
266   LD      SM400  ; Always On
      MOV     K0 U6\G4317
      MOV     K0 U6\G4417
      MOV     K0 U6\G4517
      MOV     K0 U6\G4617
      MOV     K0 U6\G4717
; Axis Ampere
295   LD      SM400  ; Always On
      MOV     U6\G2456 D7056  ; Axis 1  Ampere
      MOV     U6\G2556 D7256  ; Axis 2  Ampere
      MOV     U6\G2656 D7456  ; Axis 3  Ampere
      MOV     U6\G2756 D7656  ; Axis 4  Ampere
      MOV     U6\G2856 D7856
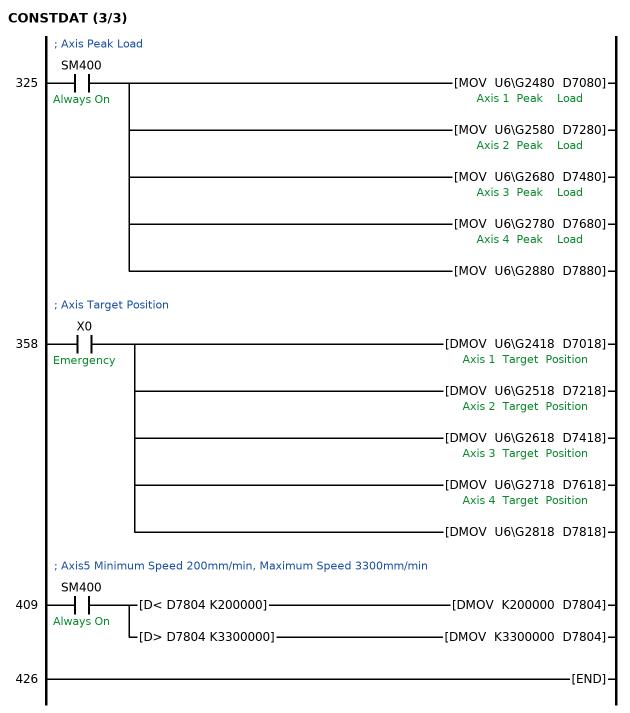
; Axis Peak Load
325   LD      SM400  ; Always On
      MOV     U6\G2480 D7080  ; Axis 1  Peak    Load
      MOV     U6\G2580 D7280  ; Axis 2  Peak    Load
      MOV     U6\G2680 D7480  ; Axis 3  Peak    Load
      MOV     U6\G2780 D7680  ; Axis 4  Peak    Load
      MOV     U6\G2880 D7880
; Axis Target Position
358   LD      X0  ; Emergency
      DMOV    U6\G2418 D7018  ; Axis 1  Target  Position
      DMOV    U6\G2518 D7218  ; Axis 2  Target  Position
      DMOV    U6\G2618 D7418  ; Axis 3  Target  Position
      DMOV    U6\G2718 D7618  ; Axis 4  Target  Position
      DMOV    U6\G2818 D7818
; Axis5 Minimum Speed 200mm/min, Maximum Speed 3300mm/min
409   LD      SM400  ; Always On
      MPS
      ANDD<   D7804 K200000
      DMOV    K200000 D7804
      MPP
      ANDD>   D7804 K3300000
      DMOV    K3300000 D7804
426   END
END_PROGRAM

PROGRAM DATA
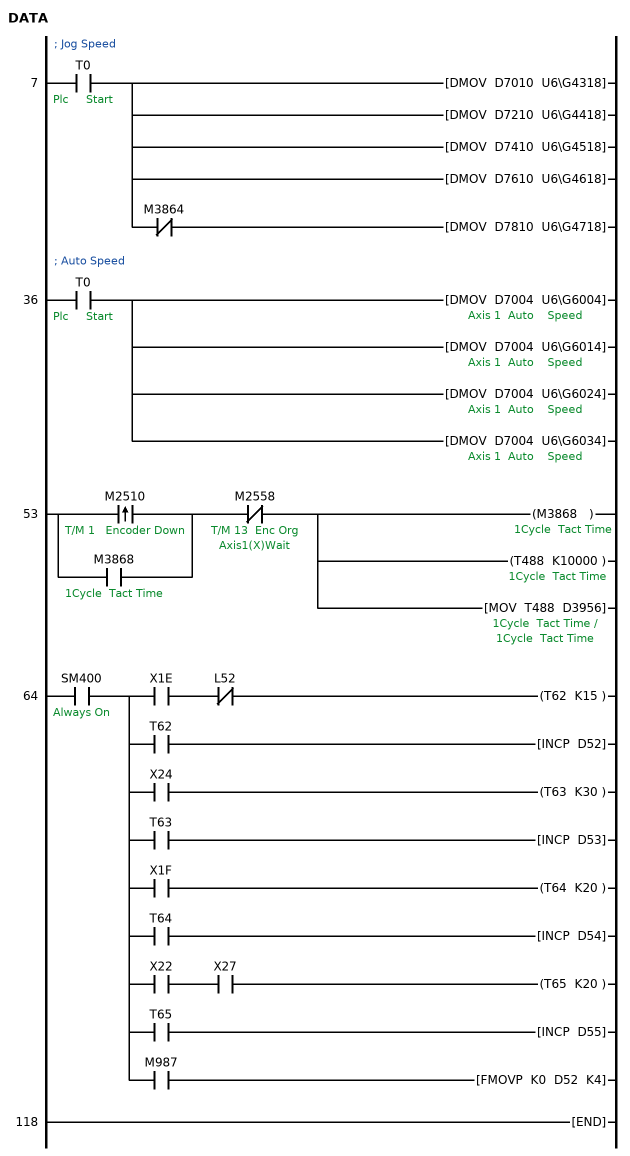
; Jog Speed
7     LD      T0  ; Plc     Start
      DMOV    D7010 U6\G4318
      DMOV    D7210 U6\G4418
      DMOV    D7410 U6\G4518
      DMOV    D7610 U6\G4618
      ANI     M3864
      DMOV    D7810 U6\G4718
; Auto Speed
36    LD      T0  ; Plc     Start
      DMOV    D7004 U6\G6004  ; Axis 1  Auto    Speed
      DMOV    D7004 U6\G6014
      DMOV    D7004 U6\G6024
      DMOV    D7004 U6\G6034
53    LDP     M2510  ; T/M 1   Encoder Down
      OR      M3868  ; 1Cycle  Tact Time
      ANI     M2558  ; T/M 13  Enc Org Axis1(X)Wait
      OUT     M3868  ; 1Cycle  Tact Time
      OUT     T488 K10000  ; 1Cycle  Tact Time
      MOV     T488 D3956  ; 1Cycle  Tact Time
64    LD      SM400  ; Always On
      MPS
      AND     X1E
      ANI     L52
      OUT     T62 K15
      MRD
      AND     T62
      INCP    D52
      MRD
      AND     X24
      OUT     T63 K30
      MRD
      AND     T63
      INCP    D53
      MRD
      AND     X1F
      OUT     T64 K20
      MRD
      AND     T64
      INCP    D54
      MRD
      AND     X22
      AND     X27
      OUT     T65 K20
      MRD
      AND     T65
      INCP    D55
      MPP
      AND     M987
      FMOVP   K0 D52 K4
118   END
END_PROGRAM

PROGRAM MANUAL
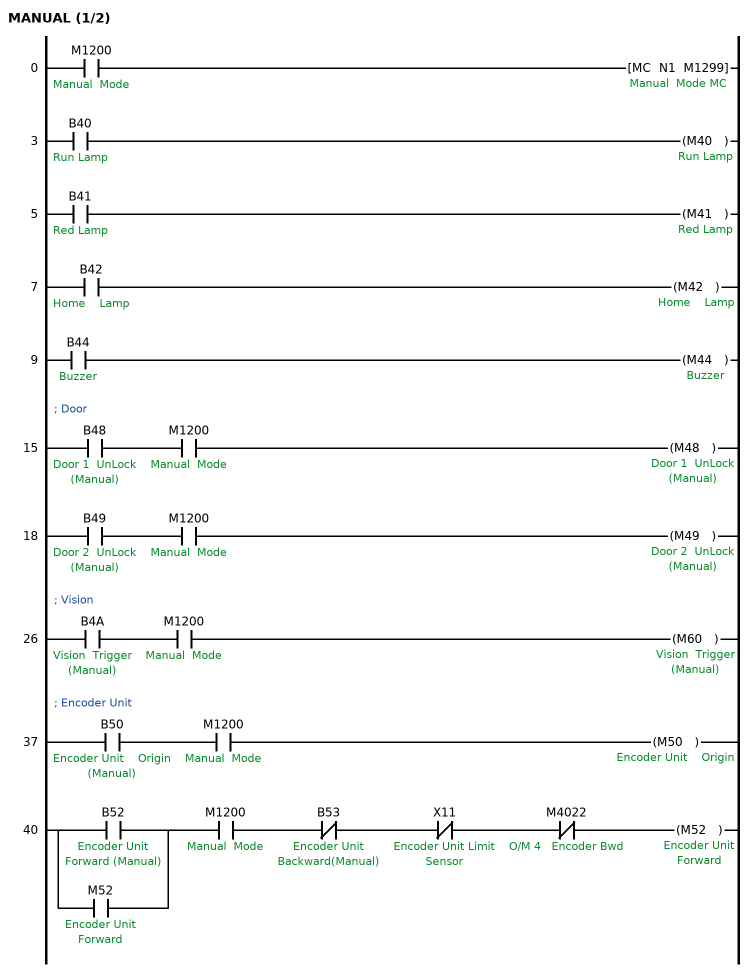
0     LD      M1200  ; Manual  Mode
      MC      N1 M1299  ; Manual  Mode MC
3     LD      B40  ; Run Lamp
      OUT     M40  ; Run Lamp
5     LD      B41  ; Red Lamp
      OUT     M41  ; Red Lamp
7     LD      B42  ; Home    Lamp
      OUT     M42  ; Home    Lamp
9     LD      B44  ; Buzzer
      OUT     M44  ; Buzzer
; Door
15    LD      B48  ; Door 1  UnLock  (Manual)
      AND     M1200  ; Manual  Mode
      OUT     M48  ; Door 1  UnLock  (Manual)
18    LD      B49  ; Door 2  UnLock  (Manual)
      AND     M1200  ; Manual  Mode
      OUT     M49  ; Door 2  UnLock  (Manual)
; Vision
26    LD      B4A  ; Vision  Trigger (Manual)
      AND     M1200  ; Manual  Mode
      OUT     M60  ; Vision  Trigger (Manual)
; Encoder Unit
37    LD      B50  ; Encoder Unit    Origin  (Manual)
      AND     M1200  ; Manual  Mode
      OUT     M50  ; Encoder Unit    Origin
40    LD      B52  ; Encoder Unit    Forward (Manual)
      OR      M52  ; Encoder Unit    Forward
      AND     M1200  ; Manual  Mode
      ANI     B53  ; Encoder Unit    Backward(Manual)
      ANI     X11  ; Encoder Unit Limit Sensor
      ANI     M4022  ; O/M 4   Encoder Bwd
      OUT     M52  ; Encoder Unit    Forward
